LIN {X 0,Y 257.714,Z 380.293,A -85,B 0,C 180,E1 -18614.986,E2 -18614.986} C_VEL
LIN {X 0,Y 256.37,Z 386.255,A -85,B 0,C 180,E1 -18617.333,E2 -18617.333} C_VEL
LIN {X 0,Y 255.344,Z 390.968,A -85,B 0,C 180,E1 -18619.695,E2 -18619.695} C_VEL
LIN {X 0,Y 254.63,Z 394.575,A -85,B 0,C 180,E1 -18622.069,E2 -18622.069} C_VEL
LIN {X 0,Y 254.242,Z 397.09,A -85,B 0,C 180,E1 -18624.356,E2 -18624.356} C_VEL
LIN {X 0,Y 254.025,Z 398.836,A -85,B 0,C 180,E1 -18626.829,E2 -18626.829} C_VEL
LIN {X 0,Y 253.97,Z 399.449,A -85,B 0,C 180,E1 -18628.415,E2 -18628.415} C_VEL
LIN {X 0,Y 253.984,Z 399.68,A -85,B 0,C 180,E1 -18630.001,E2 -18630.001} C_VEL
LIN {X 0,Y 253.969,Z 399.486,A -85,B 0,C 180,E1 -18631.586,E2 -18631.586} C_VEL
LIN {X 0,Y 254.023,Z 398.897,A -85,B 0,C 180,E1 -18633.173,E2 -18633.173} C_VEL
LIN {X 0,Y 254.332,Z 396.56,A -85,B 0,C 180,E1 -18636.347,E2 -18636.347} C_VEL
LIN {X 0,Y 254.856,Z 393.678,A -85,B 0,C 180,E1 -18638.724,E2 -18638.724} C_VEL
LIN {X 0,Y 255.623,Z 389.771,A -85,B 0,C 180,E1 -18641.097,E2 -18641.097} C_VEL
LIN {X 0,Y 256.754,Z 384.732,A -85,B 0,C 180,E1 -18643.454,E2 -18643.454} C_VEL
LIN {X 0,Y 258.236,Z 378.388,A -85,B 0,C 180,E1 -18645.793,E2 -18645.793} C_VEL
LIN {X 0,Y 260.119,Z 370.451,A -85,B 0,C 180,E1 -18648.102,E2 -18648.102} C_VEL
LIN {X 0,Y 262.191,Z 360.583,A -85,B 0,C 180,E1 -18650.394,E2 -18650.394} C_VEL
LIN {X 0,Y 264.233,Z 350.223,A -85,B 0,C 180,E1 -18652.273,E2 -18652.273} C_VEL
LIN {X 0,Y 266.512,Z 338.538,A -85,B 0,C 180,E1 -18653.919,E2 -18653.919} C_VEL
LIN {X 0,Y 268.291,Z 326.889,A -85,B 0,C 180,E1 -18655.194,E2 -18655.194} C_VEL
LIN {X 0,Y 269.794,Z 314.77,A -85,B 0,C 180,E1 -18656.181,E2 -18656.181} C_VEL
LIN {X 0,Y 270.995,Z 301.535,A -85,B 0,C 180,E1 -18656.939,E2 -18656.939} C_VEL
LIN {X 0,Y 271.629,Z 288.539,A -85,B 0,C 180,E1 -18657.391,E2 -18657.391} C_VEL
LIN {X 0,Y 273.449,Z 229.394,A -85,B 0,C 180,E1 -18658.918,E2 -18658.918} C_VEL
LIN {X 0,Y 271.728,Z 220.396,A -85,B 0,C 180,E1 -18659.386,E2 -18659.386} C_VEL
LIN {X 0,Y 264.81,Z 203.367,A -85,B 0,C 180,E1 -18660.76,E2 -18660.76} C_VEL
LIN {X 0,Y 257.854,Z 188.654,A -85,B 0,C 180,E1 -18662.208,E2 -18662.208} C_VEL
LIN {X 0,Y 256.723,Z 184.121,A -85,B 0,C 180,E1 -18664.077,E2 -18664.077} C_VEL
LIN {X 0,Y 256.131,Z 181.593,A -85,B 0,C 180,E1 -18665.365,E2 -18665.365} C_VEL
LIN {X 0,Y 256.072,Z 181.56,A -85,B 0,C 180,E1 -18669.142,E2 -18669.142} C_VEL
LIN {X 0,Y 256.062,Z 181.59,A -85,B 0,C 180,E1 -18673.327,E2 -18673.327} C_VEL
LIN {X 0,Y 256.069,Z 181.556,A -85,B 0,C 180,E1 -18677.819,E2 -18677.819} C_VEL
LIN {X 0,Y 256.071,Z 181.588,A -85,B 0,C 180,E1 -18680.858,E2 -18680.858} C_VEL
LIN {X 0,Y 256.13,Z 181.548,A -85,B 0,C 180,E1 -18682.867,E2 -18682.867} C_VEL
LIN {X 0,Y 256.067,Z 181.55,A -85,B 0,C 180,E1 -18686.707,E2 -18686.707} C_VEL
LIN {X 0,Y 256.113,Z 181.58,A -85,B 0,C 180,E1 -18690.4,E2 -18690.4} C_VEL
LIN {X 0,Y 256.169,Z 181.575,A -85,B 0,C 180,E1 -18694.87,E2 -18694.87} C_VEL
LIN {X 0,Y 256.16,Z 181.565,A -85,B 0,C 180,E1 -18699.104,E2 -18699.104} C_VEL
LIN {X 0,Y 256.277,Z 181.542,A -85,B 0,C 180,E1 -18704.083,E2 -18704.083} C_VEL
LIN {X 0,Y 256.307,Z 181.551,A -85,B 0,C 180,E1 -18708.934,E2 -18708.934} C_VEL
LIN {X 0,Y 256.537,Z 181.514,A -85,B 0,C 180,E1 -18712.127,E2 -18712.127} C_VEL
LIN {X 0,Y 256.5,Z 181.515,A -85,B 0,C 180,E1 -18716.974,E2 -18716.974} C_VEL
LIN {X 0,Y 255.921,Z 181.588,A -85,B 0,C 180,E1 -18718.288,E2 -18718.288} C_VEL
LIN {X 0,Y 254.374,Z 181.792,A -85,B 0,C 180,E1 -18719.578,E2 -18719.578} C_VEL
LIN {X 0,Y 250.591,Z 182.267,A -85,B 0,C 180,E1 -18722.171,E2 -18722.171} C_VEL
LIN {X 0,Y 249.457,Z 182.394,A -85,B 0,C 180,E1 -18723.523,E2 -18723.523} C_VEL
LIN {X 0,Y 249.335,Z 182.405,A -85,B 0,C 180,E1 -18723.982,E2 -18723.982} C_VEL
LIN {X 0,Y 249.439,Z 182.413,A -85,B 0,C 180,E1 -18728.099,E2 -18728.099} C_VEL
LIN {X 0,Y 249.185,Z 182.436,A -85,B 0,C 180,E1 -18733.04,E2 -18733.04} C_VEL
LIN {X 0,Y 249.194,Z 182.434,A -85,B 0,C 180,E1 -18736.486,E2 -18736.486} C_VEL
LIN {X 0,Y 249.079,Z 182.457,A -85,B 0,C 180,E1 -18741.519,E2 -18741.519} C_VEL
LIN {X 0,Y 249.115,Z 182.447,A -85,B 0,C 180,E1 -18745.475,E2 -18745.475} C_VEL
LIN {X 0,Y 249.071,Z 182.447,A -85,B 0,C 180,E1 -18748.989,E2 -18748.989} C_VEL
LIN {X 0,Y 249.029,Z 182.466,A -85,B 0,C 180,E1 -18752.426,E2 -18752.426} C_VEL
LIN {X 0,Y 249.028,Z 182.415,A -85,B 0,C 180,E1 -18756.346,E2 -18756.346} C_VEL
LIN {X 0,Y 249.005,Z 182.468,A -85,B 0,C 180,E1 -18760.478,E2 -18760.478} C_VEL
LIN {X 0,Y 248.986,Z 182.47,A -85,B 0,C 180,E1 -18764.883,E2 -18764.883} C_VEL
LIN {X 0,Y 249.009,Z 182.459,A -85,B 0,C 180,E1 -18767.362,E2 -18767.362} C_VEL
LIN {X 0,Y 249.027,Z 182.436,A -85,B 0,C 180,E1 -18771.62,E2 -18771.62} C_VEL
LIN {X 0,Y 249.101,Z 182.673,A -85,B 0,C 180,E1 -18772.58,E2 -18772.58} C_VEL
LIN {X 0,Y 251.278,Z 191.568,A -85,B 0,C 180,E1 -18776.62,E2 -18776.62} C_VEL
LIN {X 0,Y 251.564,Z 192.641,A -85,B 0,C 180,E1 -18776.942,E2 -18776.942} C_VEL
LIN {X 0,Y 259.446,Z 209.734,A -85,B 0,C 180,E1 -18778.65,E2 -18778.65} C_VEL
LIN {X 0,Y 264.513,Z 222.59,A -85,B 0,C 180,E1 -18779.712,E2 -18779.712} C_VEL
LIN {X 0,Y 267.062,Z 239.045,A -85,B 0,C 180,E1 -18780.529,E2 -18780.529} C_VEL
LIN {X 0,Y 264.966,Z 300.538,A -85,B 0,C 180,E1 -18782.182,E2 -18782.182} C_VEL
LIN {X 0,Y 263.782,Z 314.425,A -85,B 0,C 180,E1 -18782.854,E2 -18782.854} C_VEL
LIN {X 0,Y 262.218,Z 326.85,A -85,B 0,C 180,E1 -18783.753,E2 -18783.753} C_VEL
LIN {X 0,Y 260.587,Z 337.935,A -85,B 0,C 180,E1 -18784.863,E2 -18784.863} C_VEL
LIN {X 0,Y 258.448,Z 349.485,A -85,B 0,C 180,E1 -18786.353,E2 -18786.353} C_VEL
LIN {X 0,Y 256.294,Z 359.884,A -85,B 0,C 180,E1 -18788.061,E2 -18788.061} C_VEL
LIN {X 0,Y 254.189,Z 369.509,A -85,B 0,C 180,E1 -18790.062,E2 -18790.062} C_VEL
LIN {X 0,Y 252.306,Z 377.598,A -85,B 0,C 180,E1 -18792.157,E2 -18792.157} C_VEL
LIN {X 0,Y 250.517,Z 385.001,A -85,B 0,C 180,E1 -18794.543,E2 -18794.543} C_VEL
LIN {X 0,Y 249.061,Z 390.944,A -85,B 0,C 180,E1 -18796.953,E2 -18796.953} C_VEL
LIN {X 0,Y 248.039,Z 395.639,A -85,B 0,C 180,E1 -18799.387,E2 -18799.387} C_VEL
LIN {X 0,Y 247.375,Z 399.225,A -85,B 0,C 180,E1 -18801.833,E2 -18801.833} C_VEL
LIN {X 0,Y 247.084,Z 401.074,A -85,B 0,C 180,E1 -18803.466,E2 -18803.466} C_VEL
LIN {X 0,Y 246.923,Z 402.459,A -85,B 0,C 180,E1 -18805.101,E2 -18805.101} C_VEL
LIN {X 0,Y 246.86,Z 404.051,A -85,B 0,C 180,E1 -18808.368,E2 -18808.368} C_VEL
LIN {X 0,Y 246.891,Z 404.262,A -85,B 0,C 180,E1 -18809.999,E2 -18809.999} C_VEL
LIN {X 0,Y 246.86,Z 404.041,A -85,B 0,C 180,E1 -18811.631,E2 -18811.631} C_VEL
LIN {X 0,Y 246.924,Z 402.437,A -85,B 0,C 180,E1 -18814.897,E2 -18814.897} C_VEL
LIN {X 0,Y 247.086,Z 401.042,A -85,B 0,C 180,E1 -18816.532,E2 -18816.532} C_VEL
LIN {X 0,Y 247.563,Z 398.112,A -85,B 0,C 180,E1 -18818.982,E2 -18818.982} C_VEL
LIN {X 0,Y 248.329,Z 394.147,A -85,B 0,C 180,E1 -18821.425,E2 -18821.425} C_VEL
LIN {X 0,Y 249.704,Z 388.048,A -85,B 0,C 180,E1 -18824.256,E2 -18824.256} C_VEL
LIN {X 0,Y 251.396,Z 381.387,A -85,B 0,C 180,E1 -18826.65,E2 -18826.65} C_VEL
LIN {X 0,Y 253.374,Z 373.12,A -85,B 0,C 180,E1 -18829.02,E2 -18829.02} C_VEL
LIN {X 0,Y 255.181,Z 364.638,A -85,B 0,C 180,E1 -18830.978,E2 -18830.978} C_VEL
LIN {X 0,Y 257.424,Z 354.157,A -85,B 0,C 180,E1 -18832.894,E2 -18832.894} C_VEL
LIN {X 0,Y 259.694,Z 342.355,A -85,B 0,C 180,E1 -18834.586,E2 -18834.586} C_VEL
LIN {X 0,Y 261.675,Z 330.462,A -85,B 0,C 180,E1 -18835.875,E2 -18835.875} C_VEL
LIN {X 0,Y 263.243,Z 318.078,A -85,B 0,C 180,E1 -18836.883,E2 -18836.883} C_VEL
LIN {X 0,Y 264.56,Z 305.317,A -85,B 0,C 180,E1 -18837.594,E2 -18837.594} C_VEL
LIN {X 0,Y 265.264,Z 291.803,A -85,B 0,C 180,E1 -18838.051,E2 -18838.051} C_VEL
LIN {X 0,Y 266.926,Z 237.825,A -85,B 0,C 180,E1 -18839.482,E2 -18839.482} C_VEL
LIN {X 0,Y 264.151,Z 221.481,A -85,B 0,C 180,E1 -18840.324,E2 -18840.324} C_VEL
LIN {X 0,Y 257.7,Z 205.912,A -85,B 0,C 180,E1 -18841.661,E2 -18841.661} C_VEL
LIN {X 0,Y 251.481,Z 192.518,A -85,B 0,C 180,E1 -18843.029,E2 -18843.029} C_VEL
LIN {X 0,Y 250.518,Z 188.305,A -85,B 0,C 180,E1 -18844.751,E2 -18844.751} C_VEL
LIN {X 0,Y 249.06,Z 182.485,A -85,B 0,C 180,E1 -18847.542,E2 -18847.542} C_VEL
LIN {X 0,Y 249.002,Z 182.46,A -85,B 0,C 180,E1 -18850.477,E2 -18850.477} C_VEL
LIN {X 0,Y 248.981,Z 182.473,A -85,B 0,C 180,E1 -18854.882,E2 -18854.882} C_VEL
LIN {X 0,Y 249.004,Z 182.457,A -85,B 0,C 180,E1 -18857.36,E2 -18857.36} C_VEL
LIN {X 0,Y 249.02,Z 182.43,A -85,B 0,C 180,E1 -18861.618,E2 -18861.618} C_VEL
LIN {X 0,Y 249.037,Z 182.439,A -85,B 0,C 180,E1 -18865.638,E2 -18865.638} C_VEL
LIN {X 0,Y 249.041,Z 182.454,A -85,B 0,C 180,E1 -18869.472,E2 -18869.472} C_VEL
LIN {X 0,Y 249.061,Z 182.462,A -85,B 0,C 180,E1 -18873.161,E2 -18873.161} C_VEL
LIN {X 0,Y 249.052,Z 182.447,A -85,B 0,C 180,E1 -18876.73,E2 -18876.73} C_VEL
LIN {X 0,Y 249.082,Z 182.452,A -85,B 0,C 180,E1 -18880.209,E2 -18880.209} C_VEL
LIN {X 0,Y 249.188,Z 182.437,A -85,B 0,C 180,E1 -18883.618,E2 -18883.618} C_VEL
LIN {X 0,Y 249.243,Z 182.418,A -85,B 0,C 180,E1 -18888.616,E2 -18888.616} C_VEL
LIN {X 0,Y 249.471,Z 182.409,A -85,B 0,C 180,E1 -18891.903,E2 -18891.903} C_VEL
LIN {X 0,Y 249.422,Z 182.401,A -85,B 0,C 180,E1 -18896.769,E2 -18896.769} C_VEL
LIN {X 0,Y 249.719,Z 182.375,A -85,B 0,C 180,E1 -18900,E2 -18900} C_VEL
LIN {X 0,Y 249.423,Z 182.397,A -85,B 0,C 180,E1 -18903.231,E2 -18903.231} C_VEL
LIN {X 0,Y 249.473,Z 182.391,A -85,B 0,C 180,E1 -18908.098,E2 -18908.098} C_VEL
LIN {X 0,Y 249.244,Z 182.433,A -85,B 0,C 180,E1 -18911.384,E2 -18911.384} C_VEL
LIN {X 0,Y 249.211,Z 182.424,A -85,B 0,C 180,E1 -18916.504,E2 -18916.504} C_VEL
LIN {X 0,Y 249.08,Z 182.443,A -85,B 0,C 180,E1 -18921.519,E2 -18921.519} C_VEL
LIN {X 0,Y 249.124,Z 182.453,A -85,B 0,C 180,E1 -18925.483,E2 -18925.483} C_VEL
LIN {X 0,Y 249.077,Z 182.451,A -85,B 0,C 180,E1 -18928.994,E2 -18928.994} C_VEL
LIN {X 0,Y 249.024,Z 182.447,A -85,B 0,C 180,E1 -18932.427,E2 -18932.427} C_VEL
LIN {X 0,Y 249.024,Z 182.418,A -85,B 0,C 180,E1 -18936.347,E2 -18936.347} C_VEL
LIN {X 0,Y 249.001,Z 182.465,A -85,B 0,C 180,E1 -18940.479,E2 -18940.479} C_VEL
LIN {X 0,Y 248.988,Z 182.442,A -85,B 0,C 180,E1 -18944.883,E2 -18944.883} C_VEL
LIN {X 0,Y 249.012,Z 182.465,A -85,B 0,C 180,E1 -18947.364,E2 -18947.364} C_VEL
LIN {X 0,Y 249.041,Z 182.452,A -85,B 0,C 180,E1 -18952.202,E2 -18952.202} C_VEL
LIN {X 0,Y 249.12,Z 182.674,A -85,B 0,C 180,E1 -18954.191,E2 -18954.191} C_VEL
LIN {X 0,Y 250.596,Z 188.64,A -85,B 0,C 180,E1 -18956.872,E2 -18956.872} C_VEL
LIN {X 0,Y 257.409,Z 202.804,A -85,B 0,C 180,E1 -18958.373,E2 -18958.373} C_VEL
LIN {X 0,Y 263.323,Z 216.402,A -85,B 0,C 180,E1 -18959.587,E2 -18959.587} C_VEL
LIN {X 0,Y 266.09,Z 223.996,A -85,B 0,C 180,E1 -18960.17,E2 -18960.17} C_VEL
LIN {X 0,Y 267.251,Z 231.184,A -85,B 0,C 180,E1 -18960.531,E2 -18960.531} C_VEL
LIN {X 0,Y 265.118,Z 295.563,A -85,B 0,C 180,E1 -18962.255,E2 -18962.255} C_VEL
LIN {X 0,Y 263.939,Z 308.907,A -85,B 0,C 180,E1 -18962.873,E2 -18962.873} C_VEL
LIN {X 0,Y 262.584,Z 321.658,A -85,B 0,C 180,E1 -18963.794,E2 -18963.794} C_VEL
LIN {X 0,Y 260.868,Z 332.985,A -85,B 0,C 180,E1 -18964.894,E2 -18964.894} C_VEL
LIN {X 0,Y 258.791,Z 344.638,A -85,B 0,C 180,E1 -18966.388,E2 -18966.388} C_VEL
LIN {X 0,Y 256.651,Z 355.106,A -85,B 0,C 180,E1 -18968.094,E2 -18968.094} C_VEL
LIN {X 0,Y 254.961,Z 363.35,A -85,B 0,C 180,E1 -18969.773,E2 -18969.773} C_VEL
LIN {X 0,Y 253.136,Z 371.541,A -85,B 0,C 180,E1 -18971.801,E2 -18971.801} C_VEL
LIN {X 0,Y 251.114,Z 379.246,A -85,B 0,C 180,E1 -18974.166,E2 -18974.166} C_VEL
LIN {X 0,Y 249.445,Z 386.321,A -85,B 0,C 180,E1 -18976.975,E2 -18976.975} C_VEL
LIN {X 0,Y 248.333,Z 391.034,A -85,B 0,C 180,E1 -18979.401,E2 -18979.401} C_VEL
LIN {X 0,Y 247.602,Z 394.641,A -85,B 0,C 180,E1 -18981.842,E2 -18981.842} C_VEL
LIN {X 0,Y 247.138,Z 397.385,A -85,B 0,C 180,E1 -18984.453,E2 -18984.453} C_VEL
LIN {X 0,Y 246.931,Z 398.901,A -85,B 0,C 180,E1 -18986.738,E2 -18986.738} C_VEL
LIN {X 0,Y 246.884,Z 399.514,A -85,B 0,C 180,E1 -18988.369,E2 -18988.369} C_VEL
LIN {X 0,Y 246.894,Z 399.745,A -85,B 0,C 180,E1 -18990.001,E2 -18990.001} C_VEL
LIN {X 0,Y 246.883,Z 399.551,A -85,B 0,C 180,E1 -18991.632,E2 -18991.632} C_VEL
LIN {X 0,Y 247.06,Z 397.989,A -85,B 0,C 180,E1 -18994.896,E2 -18994.896} C_VEL
LIN {X 0,Y 247.268,Z 396.624,A -85,B 0,C 180,E1 -18996.529,E2 -18996.529} C_VEL
LIN {X 0,Y 247.831,Z 393.742,A -85,B 0,C 180,E1 -18998.973,E2 -18998.973} C_VEL
LIN {X 0,Y 248.63,Z 389.835,A -85,B 0,C 180,E1 -19001.413,E2 -19001.413} C_VEL
LIN {X 0,Y 249.818,Z 384.795,A -85,B 0,C 180,E1 -19003.835,E2 -19003.835} C_VEL
LIN {X 0,Y 251.39,Z 378.451,A -85,B 0,C 180,E1 -19006.235,E2 -19006.235} C_VEL
LIN {X 0,Y 253.358,Z 370.514,A -85,B 0,C 180,E1 -19008.603,E2 -19008.603} C_VEL
LIN {X 0,Y 255.273,Z 361.785,A -85,B 0,C 180,E1 -19010.702,E2 -19010.702} C_VEL
LIN {X 0,Y 257.45,Z 351.456,A -85,B 0,C 180,E1 -19012.681,E2 -19012.681} C_VEL
LIN {X 0,Y 259.778,Z 340.022,A -85,B 0,C 180,E1 -19014.367,E2 -19014.367} C_VEL
LIN {X 0,Y 261.58,Z 328.795,A -85,B 0,C 180,E1 -19015.673,E2 -19015.673} C_VEL
LIN {X 0,Y 263.165,Z 317.39,A -85,B 0,C 180,E1 -19016.679,E2 -19016.679} C_VEL
LIN {X 0,Y 264.491,Z 304.333,A -85,B 0,C 180,E1 -19017.496,E2 -19017.496} C_VEL
LIN {X 0,Y 265.285,Z 291.804,A -85,B 0,C 180,E1 -19017.996,E2 -19017.996} C_VEL
LIN {X 0,Y 267.208,Z 230.204,A -85,B 0,C 180,E1 -19019.637,E2 -19019.637} C_VEL
LIN {X 0,Y 265.891,Z 223.22,A -85,B 0,C 180,E1 -19020.012,E2 -19020.012} C_VEL
LIN {X 0,Y 259.258,Z 206.741,A -85,B 0,C 180,E1 -19021.387,E2 -19021.387} C_VEL
LIN {X 0,Y 251.967,Z 191.659,A -85,B 0,C 180,E1 -19022.906,E2 -19022.906} C_VEL
LIN {X 0,Y 250.562,Z 188.505,A -85,B 0,C 180,E1 -19023.302,E2 -19023.302} C_VEL
LIN {X 0,Y 249.124,Z 182.53,A -85,B 0,C 180,E1 -19026.075,E2 -19026.075} C_VEL
LIN {X 0,Y 248.992,Z 182.437,A -85,B 0,C 180,E1 -19030.481,E2 -19030.481} C_VEL
LIN {X 0,Y 249.009,Z 182.465,A -85,B 0,C 180,E1 -19032.792,E2 -19032.792} C_VEL
LIN {X 0,Y 249.009,Z 182.431,A -85,B 0,C 180,E1 -19037.361,E2 -19037.361} C_VEL
LIN {X 0,Y 249.025,Z 182.458,A -85,B 0,C 180,E1 -19041.619,E2 -19041.619} C_VEL
LIN {X 0,Y 249.042,Z 182.411,A -85,B 0,C 180,E1 -19045.639,E2 -19045.639} C_VEL
LIN {X 0,Y 249.051,Z 182.462,A -85,B 0,C 180,E1 -19049.473,E2 -19049.473} C_VEL
LIN {X 0,Y 249.068,Z 182.448,A -85,B 0,C 180,E1 -19053.161,E2 -19053.161} C_VEL
LIN {X 0,Y 249.059,Z 182.452,A -85,B 0,C 180,E1 -19056.73,E2 -19056.73} C_VEL
LIN {X 0,Y 249.106,Z 182.453,A -85,B 0,C 180,E1 -19060.211,E2 -19060.211} C_VEL
LIN {X 0,Y 249.221,Z 182.422,A -85,B 0,C 180,E1 -19063.62,E2 -19063.62} C_VEL
LIN {X 0,Y 249.25,Z 182.432,A -85,B 0,C 180,E1 -19068.616,E2 -19068.616} C_VEL
LIN {X 0,Y 249.479,Z 182.39,A -85,B 0,C 180,E1 -19071.903,E2 -19071.903} C_VEL
LIN {X 0,Y 249.428,Z 182.397,A -85,B 0,C 180,E1 -19076.769,E2 -19076.769} C_VEL
LIN {X 0,Y 249.717,Z 182.375,A -85,B 0,C 180,E1 -19080,E2 -19080} C_VEL
LIN {X 0,Y 249.426,Z 182.401,A -85,B 0,C 180,E1 -19083.23,E2 -19083.23} C_VEL
LIN {X 0,Y 249.335,Z 182.405,A -85,B 0,C 180,E1 -19083.982,E2 -19083.982} C_VEL
LIN {X 0,Y 248.59,Z 182.501,A -85,B 0,C 180,E1 -19085.332,E2 -19085.332} C_VEL
LIN {X 0,Y 245.714,Z 182.877,A -85,B 0,C 180,E1 -19087.533,E2 -19087.533} C_VEL
LIN {X 0,Y 243.307,Z 183.171,A -85,B 0,C 180,E1 -19089.325,E2 -19089.325} C_VEL
LIN {X 0,Y 242.262,Z 183.289,A -85,B 0,C 180,E1 -19090.714,E2 -19090.714} C_VEL
LIN {X 0,Y 242.167,Z 183.299,A -85,B 0,C 180,E1 -19091.185,E2 -19091.185} C_VEL
LIN {X 0,Y 242.136,Z 183.324,A -85,B 0,C 180,E1 -19095.143,E2 -19095.143} C_VEL
LIN {X 0,Y 242.051,Z 183.317,A -85,B 0,C 180,E1 -19098.626,E2 -19098.626} C_VEL
LIN {X 0,Y 242.003,Z 183.336,A -85,B 0,C 180,E1 -19102.181,E2 -19102.181} C_VEL
LIN {X 0,Y 242.065,Z 183.33,A -85,B 0,C 180,E1 -19105.838,E2 -19105.838} C_VEL
LIN {X 0,Y 242.006,Z 183.326,A -85,B 0,C 180,E1 -19109.583,E2 -19109.583} C_VEL
LIN {X 0,Y 241.979,Z 183.332,A -85,B 0,C 180,E1 -19113.493,E2 -19113.493} C_VEL
LIN {X 0,Y 241.985,Z 183.296,A -85,B 0,C 180,E1 -19117.583,E2 -19117.583} C_VEL
LIN {X 0,Y 241.933,Z 183.341,A -85,B 0,C 180,E1 -19121.923,E2 -19121.923} C_VEL
LIN {X 0,Y 241.925,Z 183.341,A -85,B 0,C 180,E1 -19126.574,E2 -19126.574} C_VEL
LIN {X 0,Y 241.974,Z 183.334,A -85,B 0,C 180,E1 -19131.409,E2 -19131.409} C_VEL
LIN {X 0,Y 242.165,Z 184.198,A -85,B 0,C 180,E1 -19132.057,E2 -19132.057} C_VEL
LIN {X 0,Y 244.206,Z 192.08,A -85,B 0,C 180,E1 -19135.73,E2 -19135.73} C_VEL
LIN {X 0,Y 245.754,Z 195.601,A -85,B 0,C 180,E1 -19136.203,E2 -19136.203} C_VEL
LIN {X 0,Y 253.217,Z 211.541,A -85,B 0,C 180,E1 -19137.848,E2 -19137.848} C_VEL
LIN {X 0,Y 258.524,Z 224.654,A -85,B 0,C 180,E1 -19139,E2 -19139} C_VEL
LIN {X 0,Y 260.875,Z 239.859,A -85,B 0,C 180,E1 -19139.785,E2 -19139.785} C_VEL
LIN {X 0,Y 258.719,Z 300.487,A -85,B 0,C 180,E1 -19141.45,E2 -19141.45} C_VEL
LIN {X 0,Y 257.502,Z 314.37,A -85,B 0,C 180,E1 -19142.135,E2 -19142.135} C_VEL
LIN {X 0,Y 255.862,Z 326.791,A -85,B 0,C 180,E1 -19143.049,E2 -19143.049} C_VEL
LIN {X 0,Y 254.18,Z 337.874,A -85,B 0,C 180,E1 -19144.184,E2 -19144.184} C_VEL
LIN {X 0,Y 251.961,Z 349.424,A -85,B 0,C 180,E1 -19145.706,E2 -19145.706} C_VEL
LIN {X 0,Y 249.696,Z 359.822,A -85,B 0,C 180,E1 -19147.45,E2 -19147.45} C_VEL
LIN {X 0,Y 247.752,Z 368.326,A -85,B 0,C 180,E1 -19149.232,E2 -19149.232} C_VEL
LIN {X 0,Y 245.894,Z 376.164,A -85,B 0,C 180,E1 -19151.244,E2 -19151.244} C_VEL
LIN {X 0,Y 243.934,Z 383.82,A -85,B 0,C 180,E1 -19153.685,E2 -19153.685} C_VEL
LIN {X 0,Y 242.11,Z 390.88,A -85,B 0,C 180,E1 -19156.571,E2 -19156.571} C_VEL
LIN {X 0,Y 241.027,Z 395.575,A -85,B 0,C 180,E1 -19159.074,E2 -19159.074} C_VEL
LIN {X 0,Y 240.328,Z 399.161,A -85,B 0,C 180,E1 -19161.592,E2 -19161.592} C_VEL
LIN {X 0,Y 240.031,Z 401.009,A -85,B 0,C 180,E1 -19163.274,E2 -19163.274} C_VEL
LIN {X 0,Y 239.836,Z 402.478,A -85,B 0,C 180,E1 -19165.081,E2 -19165.081} C_VEL
LIN {X 0,Y 239.773,Z 403.987,A -85,B 0,C 180,E1 -19168.32,E2 -19168.32} C_VEL
LIN {X 0,Y 239.804,Z 404.197,A -85,B 0,C 180,E1 -19169.999,E2 -19169.999} C_VEL
LIN {X 0,Y 239.774,Z 403.976,A -85,B 0,C 180,E1 -19171.679,E2 -19171.679} C_VEL
LIN {X 0,Y 239.844,Z 402.372,A -85,B 0,C 180,E1 -19175.042,E2 -19175.042} C_VEL
LIN {X 0,Y 240.033,Z 400.976,A -85,B 0,C 180,E1 -19176.725,E2 -19176.725} C_VEL
LIN {X 0,Y 240.542,Z 398.046,A -85,B 0,C 180,E1 -19179.246,E2 -19179.246} C_VEL
LIN {X 0,Y 241.344,Z 394.08,A -85,B 0,C 180,E1 -19181.761,E2 -19181.761} C_VEL
LIN {X 0,Y 242.787,Z 387.981,A -85,B 0,C 180,E1 -19184.671,E2 -19184.671} C_VEL
LIN {X 0,Y 244.598,Z 381.32,A -85,B 0,C 180,E1 -19187.127,E2 -19187.127} C_VEL
LIN {X 0,Y 246.664,Z 373.053,A -85,B 0,C 180,E1 -19189.558,E2 -19189.558} C_VEL
LIN {X 0,Y 248.534,Z 364.57,A -85,B 0,C 180,E1 -19191.567,E2 -19191.567} C_VEL
LIN {X 0,Y 250.886,Z 354.089,A -85,B 0,C 180,E1 -19193.526,E2 -19193.526} C_VEL
LIN {X 0,Y 253.26,Z 342.286,A -85,B 0,C 180,E1 -19195.254,E2 -19195.254} C_VEL
LIN {X 0,Y 255.3,Z 330.391,A -85,B 0,C 180,E1 -19196.571,E2 -19196.571} C_VEL
LIN {X 0,Y 256.939,Z 318.005,A -85,B 0,C 180,E1 -19197.598,E2 -19197.598} C_VEL
LIN {X 0,Y 258.3,Z 305.24,A -85,B 0,C 180,E1 -19198.322,E2 -19198.322} C_VEL
LIN {X 0,Y 259.029,Z 291.717,A -85,B 0,C 180,E1 -19198.788,E2 -19198.788} C_VEL
LIN {X 0,Y 260.752,Z 239.019,A -85,B 0,C 180,E1 -19200.212,E2 -19200.212} C_VEL
LIN {X 0,Y 258.277,Z 224.097,A -85,B 0,C 180,E1 -19201.003,E2 -19201.003} C_VEL
LIN {X 0,Y 252.02,Z 208.973,A -85,B 0,C 180,E1 -19202.357,E2 -19202.357} C_VEL
LIN {X 0,Y 245.469,Z 195.187,A -85,B 0,C 180,E1 -19203.802,E2 -19203.802} C_VEL
LIN {X 0,Y 244.197,Z 192.213,A -85,B 0,C 180,E1 -19204.192,E2 -19204.192} C_VEL
LIN {X 0,Y 242.403,Z 184.961,A -85,B 0,C 180,E1 -19207.505,E2 -19207.505} C_VEL
LIN {X 0,Y 241.989,Z 183.354,A -85,B 0,C 180,E1 -19208.424,E2 -19208.424} C_VEL
LIN {X 0,Y 241.929,Z 183.344,A -85,B 0,C 180,E1 -19211.922,E2 -19211.922} C_VEL
LIN {X 0,Y 241.92,Z 183.338,A -85,B 0,C 180,E1 -19216.572,E2 -19216.572} C_VEL
LIN {X 0,Y 241.951,Z 183.336,A -85,B 0,C 180,E1 -19220.28,E2 -19220.28} C_VEL
LIN {X 0,Y 241.975,Z 183.299,A -85,B 0,C 180,E1 -19224.487,E2 -19224.487} C_VEL
LIN {X 0,Y 241.967,Z 183.345,A -85,B 0,C 180,E1 -19228.479,E2 -19228.479} C_VEL
LIN {X 0,Y 241.994,Z 183.338,A -85,B 0,C 180,E1 -19232.311,E2 -19232.311} C_VEL
LIN {X 0,Y 242.033,Z 183.318,A -85,B 0,C 180,E1 -19236.013,E2 -19236.013} C_VEL
LIN {X 0,Y 242.016,Z 183.337,A -85,B 0,C 180,E1 -19239.606,E2 -19239.606} C_VEL
LIN {X 0,Y 242.12,Z 183.312,A -85,B 0,C 180,E1 -19243.306,E2 -19243.306} C_VEL
LIN {X 0,Y 242.176,Z 183.298,A -85,B 0,C 180,E1 -19248.279,E2 -19248.279} C_VEL
LIN {X 0,Y 242.418,Z 183.287,A -85,B 0,C 180,E1 -19251.665,E2 -19251.665} C_VEL
LIN {X 0,Y 242.245,Z 183.287,A -85,B 0,C 180,E1 -19255.007,E2 -19255.007} C_VEL
LIN {X 0,Y 242.626,Z 183.262,A -85,B 0,C 180,E1 -19258.34,E2 -19258.34} C_VEL
LIN {X 0,Y 242.626,Z 183.242,A -85,B 0,C 180,E1 -19261.66,E2 -19261.66} C_VEL
LIN {X 0,Y 242.414,Z 183.282,A -85,B 0,C 180,E1 -19266.815,E2 -19266.815} C_VEL
LIN {X 0,Y 242.306,Z 183.28,A -85,B 0,C 180,E1 -19270.022,E2 -19270.022} C_VEL
LIN {X 0,Y 242.156,Z 183.302,A -85,B 0,C 180,E1 -19275.142,E2 -19275.142} C_VEL
LIN {X 0,Y 242.066,Z 183.333,A -85,B 0,C 180,E1 -19278.625,E2 -19278.625} C_VEL
LIN {X 0,Y 242.006,Z 183.322,A -85,B 0,C 180,E1 -19282.181,E2 -19282.181} C_VEL
LIN {X 0,Y 242.06,Z 183.33,A -85,B 0,C 180,E1 -19285.839,E2 -19285.839} C_VEL
LIN {X 0,Y 242.024,Z 183.334,A -85,B 0,C 180,E1 -19289.581,E2 -19289.581} C_VEL
LIN {X 0,Y 241.975,Z 183.302,A -85,B 0,C 180,E1 -19293.494,E2 -19293.494} C_VEL
LIN {X 0,Y 241.981,Z 183.314,A -85,B 0,C 180,E1 -19297.584,E2 -19297.584} C_VEL
LIN {X 0,Y 241.929,Z 183.321,A -85,B 0,C 180,E1 -19301.925,E2 -19301.925} C_VEL
LIN {X 0,Y 241.929,Z 183.35,A -85,B 0,C 180,E1 -19306.573,E2 -19306.573} C_VEL
LIN {X 0,Y 241.993,Z 183.319,A -85,B 0,C 180,E1 -19311.642,E2 -19311.642} C_VEL
LIN {X 0,Y 242.064,Z 183.552,A -85,B 0,C 180,E1 -19313.337,E2 -19313.337} C_VEL
LIN {X 0,Y 243.357,Z 188.803,A -85,B 0,C 180,E1 -19315.768,E2 -19315.768} C_VEL
LIN {X 0,Y 249.859,Z 201.93,A -85,B 0,C 180,E1 -19317.268,E2 -19317.268} C_VEL
LIN {X 0,Y 256.236,Z 216.029,A -85,B 0,C 180,E1 -19318.637,E2 -19318.637} C_VEL
LIN {X 0,Y 260.178,Z 226.549,A -85,B 0,C 180,E1 -19319.498,E2 -19319.498} C_VEL
LIN {X 0,Y 261.071,Z 232.307,A -85,B 0,C 180,E1 -19319.794,E2 -19319.794} C_VEL
LIN {X 0,Y 258.877,Z 295.646,A -85,B 0,C 180,E1 -19321.526,E2 -19321.526} C_VEL
LIN {X 0,Y 257.656,Z 308.982,A -85,B 0,C 180,E1 -19322.154,E2 -19322.154} C_VEL
LIN {X 0,Y 256.243,Z 321.73,A -85,B 0,C 180,E1 -19323.094,E2 -19323.094} C_VEL
LIN {X 0,Y 254.448,Z 333.055,A -85,B 0,C 180,E1 -19324.215,E2 -19324.215} C_VEL
LIN {X 0,Y 252.289,Z 344.707,A -85,B 0,C 180,E1 -19325.741,E2 -19325.741} C_VEL
LIN {X 0,Y 250.08,Z 355.174,A -85,B 0,C 180,E1 -19327.488,E2 -19327.488} C_VEL
LIN {X 0,Y 248.162,Z 364.038,A -85,B 0,C 180,E1 -19329.345,E2 -19329.345} C_VEL
LIN {X 0,Y 246.025,Z 372.998,A -85,B 0,C 180,E1 -19331.687,E2 -19331.687} C_VEL
LIN {X 0,Y 243.983,Z 380.427,A -85,B 0,C 180,E1 -19334.12,E2 -19334.12} C_VEL
LIN {X 0,Y 242.514,Z 386.388,A -85,B 0,C 180,E1 -19336.596,E2 -19336.596} C_VEL
LIN {X 0,Y 241.341,Z 391.1,A -85,B 0,C 180,E1 -19339.09,E2 -19339.09} C_VEL
LIN {X 0,Y 240.556,Z 394.707,A -85,B 0,C 180,E1 -19341.601,E2 -19341.601} C_VEL
LIN {X 0,Y 240.025,Z 397.702,A -85,B 0,C 180,E1 -19344.583,E2 -19344.583} C_VEL
LIN {X 0,Y 239.841,Z 398.967,A -85,B 0,C 180,E1 -19346.641,E2 -19346.641} C_VEL
LIN {X 0,Y 239.8,Z 399.579,A -85,B 0,C 180,E1 -19348.321,E2 -19348.321} C_VEL
LIN {X 0,Y 239.807,Z 399.81,A -85,B 0,C 180,E1 -19350.001,E2 -19350.001} C_VEL
LIN {X 0,Y 239.799,Z 399.615,A -85,B 0,C 180,E1 -19351.68,E2 -19351.68} C_VEL
LIN {X 0,Y 239.97,Z 398.053,A -85,B 0,C 180,E1 -19355.041,E2 -19355.041} C_VEL
LIN {X 0,Y 240.205,Z 396.689,A -85,B 0,C 180,E1 -19356.721,E2 -19356.721} C_VEL
LIN {X 0,Y 240.794,Z 393.806,A -85,B 0,C 180,E1 -19359.238,E2 -19359.238} C_VEL
LIN {X 0,Y 241.661,Z 389.899,A -85,B 0,C 180,E1 -19361.746,E2 -19361.746} C_VEL
LIN {X 0,Y 242.904,Z 384.859,A -85,B 0,C 180,E1 -19364.237,E2 -19364.237} C_VEL
LIN {X 0,Y 244.571,Z 378.514,A -85,B 0,C 180,E1 -19366.7,E2 -19366.7} C_VEL
LIN {X 0,Y 246.618,Z 370.577,A -85,B 0,C 180,E1 -19369.131,E2 -19369.131} C_VEL
LIN {X 0,Y 248.56,Z 362.147,A -85,B 0,C 180,E1 -19371.214,E2 -19371.214} C_VEL
LIN {X 0,Y 250.685,Z 352.618,A -85,B 0,C 180,E1 -19373.11,E2 -19373.11} C_VEL
LIN {X 0,Y 253.017,Z 341.508,A -85,B 0,C 180,E1 -19374.843,E2 -19374.843} C_VEL
LIN {X 0,Y 255.215,Z 328.854,A -85,B 0,C 180,E1 -19376.362,E2 -19376.362} C_VEL
LIN {X 0,Y 256.984,Z 316.183,A -85,B 0,C 180,E1 -19377.484,E2 -19377.484} C_VEL
LIN {X 0,Y 258.288,Z 303.471,A -85,B 0,C 180,E1 -19378.27,E2 -19378.27} C_VEL
LIN {X 0,Y 259.107,Z 290.345,A -85,B 0,C 180,E1 -19378.78,E2 -19378.78} C_VEL
LIN {X 0,Y 261.055,Z 231.321,A -85,B 0,C 180,E1 -19380.375,E2 -19380.375} C_VEL
LIN {X 0,Y 259.856,Z 225.337,A -85,B 0,C 180,E1 -19380.718,E2 -19380.718} C_VEL
LIN {X 0,Y 253.661,Z 209.944,A -85,B 0,C 180,E1 -19382.057,E2 -19382.057} C_VEL
LIN {X 0,Y 246.715,Z 195.495,A -85,B 0,C 180,E1 -19383.568,E2 -19383.568} C_VEL
LIN {X 0,Y 243.35,Z 188.71,A -85,B 0,C 180,E1 -19384.397,E2 -19384.397} C_VEL
LIN {X 0,Y 242.076,Z 183.57,A -85,B 0,C 180,E1 -19386.801,E2 -19386.801} C_VEL
LIN {X 0,Y 241.949,Z 183.314,A -85,B 0,C 180,E1 -19389.72,E2 -19389.72} C_VEL
LIN {X 0,Y 241.926,Z 183.34,A -85,B 0,C 180,E1 -19394.203,E2 -19394.203} C_VEL
LIN {X 0,Y 241.933,Z 183.318,A -85,B 0,C 180,E1 -19398.076,E2 -19398.076} C_VEL
LIN {X 0,Y 241.985,Z 183.317,A -85,B 0,C 180,E1 -19402.417,E2 -19402.417} C_VEL
LIN {X 0,Y 241.98,Z 183.299,A -85,B 0,C 180,E1 -19406.507,E2 -19406.507} C_VEL
LIN {X 0,Y 242.036,Z 183.333,A -85,B 0,C 180,E1 -19410.587,E2 -19410.587} C_VEL
LIN {X 0,Y 242.067,Z 183.328,A -85,B 0,C 180,E1 -19414.183,E2 -19414.183} C_VEL
LIN {X 0,Y 242.024,Z 183.32,A -85,B 0,C 180,E1 -19418.313,E2 -19418.313} C_VEL
LIN {X 0,Y 242.162,Z 183.304,A -85,B 0,C 180,E1 -19423.278,E2 -19423.278} C_VEL
LIN {X 0,Y 242.184,Z 183.313,A -85,B 0,C 180,E1 -19428.28,E2 -19428.28} C_VEL
LIN {X 0,Y 242.425,Z 183.266,A -85,B 0,C 180,E1 -19431.665,E2 -19431.665} C_VEL
LIN {X 0,Y 242.252,Z 183.307,A -85,B 0,C 180,E1 -19435.007,E2 -19435.007} C_VEL
LIN {X 0,Y 242.632,Z 183.241,A -85,B 0,C 180,E1 -19438.34,E2 -19438.34} C_VEL
LIN {X 0,Y 242.631,Z 183.261,A -85,B 0,C 180,E1 -19441.66,E2 -19441.66} C_VEL
LIN {X 0,Y 242.412,Z 183.283,A -85,B 0,C 180,E1 -19446.659,E2 -19446.659} C_VEL
LIN {X 0,Y 242.258,Z 183.296,A -85,B 0,C 180,E1 -19450.024,E2 -19450.024} C_VEL
LIN {X 0,Y 242.167,Z 183.299,A -85,B 0,C 180,E1 -19451.185,E2 -19451.185} C_VEL
LIN {X 0,Y 241.462,Z 183.393,A -85,B 0,C 180,E1 -19452.574,E2 -19452.574} C_VEL
LIN {X 0,Y 238.564,Z 183.769,A -85,B 0,C 180,E1 -19454.836,E2 -19454.836} C_VEL
LIN {X 0,Y 236.118,Z 184.061,A -85,B 0,C 180,E1 -19456.68,E2 -19456.68} C_VEL
LIN {X 0,Y 235.069,Z 184.184,A -85,B 0,C 180,E1 -19458.112,E2 -19458.112} C_VEL
LIN {X 0,Y 234.983,Z 184.197,A -85,B 0,C 180,E1 -19458.598,E2 -19458.598} C_VEL
LIN {X 0,Y 234.95,Z 184.205,A -85,B 0,C 180,E1 -19462.884,E2 -19462.884} C_VEL
LIN {X 0,Y 234.966,Z 184.217,A -85,B 0,C 180,E1 -19466.658,E2 -19466.658} C_VEL
LIN {X 0,Y 234.921,Z 184.214,A -85,B 0,C 180,E1 -19470.569,E2 -19470.569} C_VEL
LIN {X 0,Y 234.926,Z 184.186,A -85,B 0,C 180,E1 -19474.639,E2 -19474.639} C_VEL
LIN {X 0,Y 234.941,Z 184.193,A -85,B 0,C 180,E1 -19478.945,E2 -19478.945} C_VEL
LIN {X 0,Y 234.878,Z 184.215,A -85,B 0,C 180,E1 -19483.488,E2 -19483.488} C_VEL
LIN {X 0,Y 234.878,Z 184.219,A -85,B 0,C 180,E1 -19486.512,E2 -19486.512} C_VEL
LIN {X 0,Y 234.928,Z 184.304,A -85,B 0,C 180,E1 -19490.668,E2 -19490.668} C_VEL
LIN {X 0,Y 236.783,Z 191.397,A -85,B 0,C 180,E1 -19494.27,E2 -19494.27} C_VEL
LIN {X 0,Y 237.045,Z 192.421,A -85,B 0,C 180,E1 -19494.619,E2 -19494.619} C_VEL
LIN {X 0,Y 241.553,Z 201.579,A -85,B 0,C 180,E1 -19495.745,E2 -19495.745} C_VEL
LIN {X 0,Y 248.641,Z 217.011,A -85,B 0,C 180,E1 -19497.368,E2 -19497.368} C_VEL
LIN {X 0,Y 252.725,Z 227.313,A -85,B 0,C 180,E1 -19498.295,E2 -19498.295} C_VEL
LIN {X 0,Y 254.73,Z 240.01,A -85,B 0,C 180,E1 -19498.983,E2 -19498.983} C_VEL
LIN {X 0,Y 252.517,Z 300.435,A -85,B 0,C 180,E1 -19500.681,E2 -19500.681} C_VEL
LIN {X 0,Y 251.258,Z 314.314,A -85,B 0,C 180,E1 -19501.379,E2 -19501.379} C_VEL
LIN {X 0,Y 249.552,Z 326.732,A -85,B 0,C 180,E1 -19502.31,E2 -19502.31} C_VEL
LIN {X 0,Y 247.816,Z 337.814,A -85,B 0,C 180,E1 -19503.47,E2 -19503.47} C_VEL
LIN {X 0,Y 245.496,Z 349.362,A -85,B 0,C 180,E1 -19505.023,E2 -19505.023} C_VEL
LIN {X 0,Y 243.124,Z 359.76,A -85,B 0,C 180,E1 -19506.805,E2 -19506.805} C_VEL
LIN {X 0,Y 241.01,Z 368.611,A -85,B 0,C 180,E1 -19508.712,E2 -19508.712} C_VEL
LIN {X 0,Y 238.781,Z 377.471,A -85,B 0,C 180,E1 -19511.109,E2 -19511.109} C_VEL
LIN {X 0,Y 236.815,Z 384.874,A -85,B 0,C 180,E1 -19513.624,E2 -19513.624} C_VEL
LIN {X 0,Y 235.175,Z 390.816,A -85,B 0,C 180,E1 -19516.168,E2 -19516.168} C_VEL
LIN {X 0,Y 234.03,Z 395.511,A -85,B 0,C 180,E1 -19518.743,E2 -19518.743} C_VEL
LIN {X 0,Y 233.284,Z 399.097,A -85,B 0,C 180,E1 -19521.336,E2 -19521.336} C_VEL
LIN {X 0,Y 232.977,Z 400.945,A -85,B 0,C 180,E1 -19523.069,E2 -19523.069} C_VEL
LIN {X 0,Y 232.713,Z 402.643,A -85,B 0,C 180,E1 -19525.283,E2 -19525.283} C_VEL
LIN {X 0,Y 232.67,Z 403.922,A -85,B 0,C 180,E1 -19528.268,E2 -19528.268} C_VEL
LIN {X 0,Y 232.718,Z 404.133,A -85,B 0,C 180,E1 -19529.999,E2 -19529.999} C_VEL
LIN {X 0,Y 232.671,Z 403.911,A -85,B 0,C 180,E1 -19531.73,E2 -19531.73} C_VEL
LIN {X 0,Y 232.768,Z 402.306,A -85,B 0,C 180,E1 -19535.196,E2 -19535.196} C_VEL
LIN {X 0,Y 232.978,Z 400.91,A -85,B 0,C 180,E1 -19536.929,E2 -19536.929} C_VEL
LIN {X 0,Y 233.506,Z 397.98,A -85,B 0,C 180,E1 -19539.527,E2 -19539.527} C_VEL
LIN {X 0,Y 234.377,Z 394.014,A -85,B 0,C 180,E1 -19542.115,E2 -19542.115} C_VEL
LIN {X 0,Y 235.901,Z 387.914,A -85,B 0,C 180,E1 -19545.109,E2 -19545.109} C_VEL
LIN {X 0,Y 237.814,Z 381.253,A -85,B 0,C 180,E1 -19547.631,E2 -19547.631} C_VEL
LIN {X 0,Y 239.956,Z 373.026,A -85,B 0,C 180,E1 -19550.116,E2 -19550.116} C_VEL
LIN {X 0,Y 241.919,Z 364.502,A -85,B 0,C 180,E1 -19552.188,E2 -19552.188} C_VEL
LIN {X 0,Y 244.389,Z 354.02,A -85,B 0,C 180,E1 -19554.19,E2 -19554.19} C_VEL
LIN {X 0,Y 246.85,Z 342.216,A -85,B 0,C 180,E1 -19555.958,E2 -19555.958} C_VEL
LIN {X 0,Y 248.98,Z 330.32,A -85,B 0,C 180,E1 -19557.301,E2 -19557.301} C_VEL
LIN {X 0,Y 250.685,Z 317.933,A -85,B 0,C 180,E1 -19558.348,E2 -19558.348} C_VEL
LIN {X 0,Y 252.081,Z 305.163,A -85,B 0,C 180,E1 -19559.087,E2 -19559.087} C_VEL
LIN {X 0,Y 252.834,Z 291.631,A -85,B 0,C 180,E1 -19559.562,E2 -19559.562} C_VEL
LIN {X 0,Y 254.633,Z 240.043,A -85,B 0,C 180,E1 -19560.981,E2 -19560.981} C_VEL
LIN {X 0,Y 252.474,Z 226.782,A -85,B 0,C 180,E1 -19561.707,E2 -19561.707} C_VEL
LIN {X 0,Y 246.851,Z 213.008,A -85,B 0,C 180,E1 -19562.981,E2 -19562.981} C_VEL
LIN {X 0,Y 240.165,Z 198.888,A -85,B 0,C 180,E1 -19564.519,E2 -19564.519} C_VEL
LIN {X 0,Y 236.998,Z 192.193,A -85,B 0,C 180,E1 -19565.365,E2 -19565.365} C_VEL
LIN {X 0,Y 234.999,Z 184.749,A -85,B 0,C 180,E1 -19568.961,E2 -19568.961} C_VEL
LIN {X 0,Y 234.917,Z 184.214,A -85,B 0,C 180,E1 -19569.471,E2 -19569.471} C_VEL
LIN {X 0,Y 234.88,Z 184.224,A -85,B 0,C 180,E1 -19574.1,E2 -19574.1} C_VEL
LIN {X 0,Y 234.877,Z 184.228,A -85,B 0,C 180,E1 -19578.831,E2 -19578.831} C_VEL
LIN {X 0,Y 234.912,Z 184.194,A -85,B 0,C 180,E1 -19581.077,E2 -19581.077} C_VEL
LIN {X 0,Y 234.921,Z 184.189,A -85,B 0,C 180,E1 -19585.36,E2 -19585.36} C_VEL
LIN {X 0,Y 234.916,Z 184.213,A -85,B 0,C 180,E1 -19589.43,E2 -19589.43} C_VEL
LIN {X 0,Y 234.987,Z 184.213,A -85,B 0,C 180,E1 -19593.793,E2 -19593.793} C_VEL
LIN {X 0,Y 234.984,Z 184.216,A -85,B 0,C 180,E1 -19598.967,E2 -19598.967} C_VEL
LIN {X 0,Y 235.056,Z 184.189,A -85,B 0,C 180,E1 -19603.085,E2 -19603.085} C_VEL
LIN {X 0,Y 235.106,Z 184.179,A -85,B 0,C 180,E1 -19607.922,E2 -19607.922} C_VEL
LIN {X 0,Y 235.367,Z 184.166,A -85,B 0,C 180,E1 -19611.414,E2 -19611.414} C_VEL
LIN {X 0,Y 235.393,Z 184.158,A -85,B 0,C 180,E1 -19613.141,E2 -19613.141} C_VEL
LIN {X 0,Y 235.586,Z 184.138,A -85,B 0,C 180,E1 -19618.291,E2 -19618.291} C_VEL
LIN {X 0,Y 235.586,Z 184.118,A -85,B 0,C 180,E1 -19621.71,E2 -19621.71} C_VEL
LIN {X 0,Y 235.395,Z 184.157,A -85,B 0,C 180,E1 -19626.859,E2 -19626.859} C_VEL
LIN {X 0,Y 235.23,Z 184.164,A -85,B 0,C 180,E1 -19630.327,E2 -19630.327} C_VEL
LIN {X 0,Y 235.104,Z 184.178,A -85,B 0,C 180,E1 -19635.607,E2 -19635.607} C_VEL
LIN {X 0,Y 235.001,Z 184.212,A -85,B 0,C 180,E1 -19639.206,E2 -19639.206} C_VEL
LIN {X 0,Y 234.954,Z 184.203,A -85,B 0,C 180,E1 -19642.884,E2 -19642.884} C_VEL
LIN {X 0,Y 234.963,Z 184.207,A -85,B 0,C 180,E1 -19646.658,E2 -19646.658} C_VEL
LIN {X 0,Y 234.926,Z 184.222,A -85,B 0,C 180,E1 -19650.569,E2 -19650.569} C_VEL
LIN {X 0,Y 234.921,Z 184.168,A -85,B 0,C 180,E1 -19654.64,E2 -19654.64} C_VEL
LIN {X 0,Y 234.937,Z 184.217,A -85,B 0,C 180,E1 -19658.946,E2 -19658.946} C_VEL
LIN {X 0,Y 234.875,Z 184.188,A -85,B 0,C 180,E1 -19663.489,E2 -19663.489} C_VEL
LIN {X 0,Y 234.881,Z 184.226,A -85,B 0,C 180,E1 -19666.515,E2 -19666.515} C_VEL
LIN {X 0,Y 234.914,Z 184.193,A -85,B 0,C 180,E1 -19671.08,E2 -19671.08} C_VEL
LIN {X 0,Y 235.003,Z 184.493,A -85,B 0,C 180,E1 -19672.461,E2 -19672.461} C_VEL
LIN {X 0,Y 236.142,Z 188.708,A -85,B 0,C 180,E1 -19674.528,E2 -19674.528} C_VEL
LIN {X 0,Y 237.967,Z 192.498,A -85,B 0,C 180,E1 -19675.061,E2 -19675.061} C_VEL
LIN {X 0,Y 245.923,Z 208.497,A -85,B 0,C 180,E1 -19676.899,E2 -19676.899} C_VEL
LIN {X 0,Y 251.19,Z 220.576,A -85,B 0,C 180,E1 -19678.081,E2 -19678.081} C_VEL
LIN {X 0,Y 254.289,Z 229.084,A -85,B 0,C 180,E1 -19678.792,E2 -19678.792} C_VEL
LIN {X 0,Y 254.895,Z 233.595,A -85,B 0,C 180,E1 -19679.021,E2 -19679.021} C_VEL
LIN {X 0,Y 252.605,Z 296.374,A -85,B 0,C 180,E1 -19680.784,E2 -19680.784} C_VEL
LIN {X 0,Y 251.341,Z 309.89,A -85,B 0,C 180,E1 -19681.454,E2 -19681.454} C_VEL
LIN {X 0,Y 249.779,Z 322.891,A -85,B 0,C 180,E1 -19682.453,E2 -19682.453} C_VEL
LIN {X 0,Y 247.783,Z 334.71,A -85,B 0,C 180,E1 -19683.695,E2 -19683.695} C_VEL
LIN {X 0,Y 245.58,Z 346.066,A -85,B 0,C 180,E1 -19685.259,E2 -19685.259} C_VEL
LIN {X 0,Y 243.297,Z 356.301,A -85,B 0,C 180,E1 -19687.049,E2 -19687.049} C_VEL
LIN {X 0,Y 241.079,Z 365.899,A -85,B 0,C 180,E1 -19689.191,E2 -19689.191} C_VEL
LIN {X 0,Y 238.91,Z 374.417,A -85,B 0,C 180,E1 -19691.566,E2 -19691.566} C_VEL
LIN {X 0,Y 236.884,Z 381.607,A -85,B 0,C 180,E1 -19694.073,E2 -19694.073} C_VEL
LIN {X 0,Y 235.596,Z 386.455,A -85,B 0,C 180,E1 -19696.195,E2 -19696.195} C_VEL
LIN {X 0,Y 234.366,Z 391.167,A -85,B 0,C 180,E1 -19698.761,E2 -19698.761} C_VEL
LIN {X 0,Y 233.518,Z 394.773,A -85,B 0,C 180,E1 -19701.346,E2 -19701.346} C_VEL
LIN {X 0,Y 233.164,Z 396.635,A -85,B 0,C 180,E1 -19703.076,E2 -19703.076} C_VEL
LIN {X 0,Y 232.921,Z 398.036,A -85,B 0,C 180,E1 -19704.807,E2 -19704.807} C_VEL
LIN {X 0,Y 232.699,Z 399.644,A -85,B 0,C 180,E1 -19708.27,E2 -19708.27} C_VEL
LIN {X 0,Y 232.722,Z 399.874,A -85,B 0,C 180,E1 -19710.001,E2 -19710.001} C_VEL
LIN {X 0,Y 232.698,Z 399.68,A -85,B 0,C 180,E1 -19711.731,E2 -19711.731} C_VEL
LIN {X 0,Y 232.902,Z 398.118,A -85,B 0,C 180,E1 -19715.195,E2 -19715.195} C_VEL
LIN {X 0,Y 233.136,Z 396.753,A -85,B 0,C 180,E1 -19716.926,E2 -19716.926} C_VEL
LIN {X 0,Y 233.779,Z 393.87,A -85,B 0,C 180,E1 -19719.518,E2 -19719.518} C_VEL
LIN {X 0,Y 234.708,Z 389.962,A -85,B 0,C 180,E1 -19722.1,E2 -19722.1} C_VEL
LIN {X 0,Y 236.011,Z 384.923,A -85,B 0,C 180,E1 -19724.662,E2 -19724.662} C_VEL
LIN {X 0,Y 237.773,Z 378.577,A -85,B 0,C 180,E1 -19727.192,E2 -19727.192} C_VEL
LIN {X 0,Y 239.883,Z 370.639,A -85,B 0,C 180,E1 -19729.69,E2 -19729.69} C_VEL
LIN {X 0,Y 242.302,Z 360.769,A -85,B 0,C 180,E1 -19732.152,E2 -19732.152} C_VEL
LIN {X 0,Y 244.67,Z 350.406,A -85,B 0,C 180,E1 -19734.162,E2 -19734.162} C_VEL
LIN {X 0,Y 246.937,Z 340.143,A -85,B 0,C 180,E1 -19735.723,E2 -19735.723} C_VEL
LIN {X 0,Y 248.888,Z 328.913,A -85,B 0,C 180,E1 -19737.086,E2 -19737.086} C_VEL
LIN {X 0,Y 250.713,Z 316.239,A -85,B 0,C 180,E1 -19738.232,E2 -19738.232} C_VEL
LIN {X 0,Y 252.066,Z 303.523,A -85,B 0,C 180,E1 -19739.033,E2 -19739.033} C_VEL
LIN {X 0,Y 252.917,Z 290.389,A -85,B 0,C 180,E1 -19739.553,E2 -19739.553} C_VEL
LIN {X 0,Y 254.963,Z 233.058,A -85,B 0,C 180,E1 -19741.126,E2 -19741.126} C_VEL
LIN {X 0,Y 253.993,Z 227.765,A -85,B 0,C 180,E1 -19741.43,E2 -19741.43} C_VEL
LIN {X 0,Y 247.617,Z 212.119,A -85,B 0,C 180,E1 -19742.865,E2 -19742.865} C_VEL
LIN {X 0,Y 241.484,Z 199.32,A -85,B 0,C 180,E1 -19744.262,E2 -19744.262} C_VEL
LIN {X 0,Y 236.193,Z 188.911,A -85,B 0,C 180,E1 -19745.577,E2 -19745.577} C_VEL
LIN {X 0,Y 235.231,Z 185.355,A -85,B 0,C 180,E1 -19747.229,E2 -19747.229} C_VEL
LIN {X 0,Y 234.983,Z 184.239,A -85,B 0,C 180,E1 -19747.951,E2 -19747.951} C_VEL
LIN {X 0,Y 234.877,Z 184.204,A -85,B 0,C 180,E1 -19751.578,E2 -19751.578} C_VEL
LIN {X 0,Y 234.887,Z 184.19,A -85,B 0,C 180,E1 -19755.897,E2 -19755.897} C_VEL
LIN {X 0,Y 234.881,Z 184.207,A -85,B 0,C 180,E1 -19758.831,E2 -19758.831} C_VEL
LIN {X 0,Y 234.918,Z 184.222,A -85,B 0,C 180,E1 -19761.078,E2 -19761.078} C_VEL
LIN {X 0,Y 234.926,Z 184.166,A -85,B 0,C 180,E1 -19765.361,E2 -19765.361} C_VEL
LIN {X 0,Y 234.931,Z 184.221,A -85,B 0,C 180,E1 -19769.432,E2 -19769.432} C_VEL
LIN {X 0,Y 234.993,Z 184.205,A -85,B 0,C 180,E1 -19773.794,E2 -19773.794} C_VEL
LIN {X 0,Y 234.996,Z 184.198,A -85,B 0,C 180,E1 -19778.968,E2 -19778.968} C_VEL
LIN {X 0,Y 235.094,Z 184.186,A -85,B 0,C 180,E1 -19783.06,E2 -19783.06} C_VEL
LIN {X 0,Y 235.144,Z 184.192,A -85,B 0,C 180,E1 -19787.923,E2 -19787.923} C_VEL
LIN {X 0,Y 235.375,Z 184.142,A -85,B 0,C 180,E1 -19791.414,E2 -19791.414} C_VEL
LIN {X 0,Y 235.401,Z 184.156,A -85,B 0,C 180,E1 -19793.141,E2 -19793.141} C_VEL
LIN {X 0,Y 235.591,Z 184.117,A -85,B 0,C 180,E1 -19798.29,E2 -19798.29} C_VEL
LIN {X 0,Y 235.591,Z 184.138,A -85,B 0,C 180,E1 -19801.709,E2 -19801.709} C_VEL
LIN {X 0,Y 235.362,Z 184.162,A -85,B 0,C 180,E1 -19806.86,E2 -19806.86} C_VEL
LIN {X 0,Y 235.183,Z 184.173,A -85,B 0,C 180,E1 -19810.329,E2 -19810.329} C_VEL
LIN {X 0,Y 235.083,Z 184.198,A -85,B 0,C 180,E1 -19815.608,E2 -19815.608} C_VEL
LIN {X 0,Y 234.983,Z 184.197,A -85,B 0,C 180,E1 -19818.598,E2 -19818.598} C_VEL
LIN {X 0,Y 234.305,Z 184.296,A -85,B 0,C 180,E1 -19820.029,E2 -19820.029} C_VEL
LIN {X 0,Y 231.431,Z 184.649,A -85,B 0,C 180,E1 -19822.363,E2 -19822.363} C_VEL
LIN {X 0,Y 229.008,Z 184.949,A -85,B 0,C 180,E1 -19824.266,E2 -19824.266} C_VEL
LIN {X 0,Y 227.995,Z 185.08,A -85,B 0,C 180,E1 -19825.744,E2 -19825.744} C_VEL
LIN {X 0,Y 227.926,Z 185.091,A -85,B 0,C 180,E1 -19826.245,E2 -19826.245} C_VEL
LIN {X 0,Y 227.896,Z 185.086,A -85,B 0,C 180,E1 -19830.291,E2 -19830.291} C_VEL
LIN {X 0,Y 227.876,Z 185.081,A -85,B 0,C 180,E1 -19833.721,E2 -19833.721} C_VEL
LIN {X 0,Y 227.842,Z 185.061,A -85,B 0,C 180,E1 -19838.091,E2 -19838.091} C_VEL
LIN {X 0,Y 227.805,Z 185.095,A -85,B 0,C 180,E1 -19842.744,E2 -19842.744} C_VEL
LIN {X 0,Y 227.806,Z 185.099,A -85,B 0,C 180,E1 -19847.257,E2 -19847.257} C_VEL
LIN {X 0,Y 227.906,Z 185.276,A -85,B 0,C 180,E1 -19849.758,E2 -19849.758} C_VEL
LIN {X 0,Y 229.766,Z 192.122,A -85,B 0,C 180,E1 -19853.286,E2 -19853.286} C_VEL
LIN {X 0,Y 233.141,Z 199.006,A -85,B 0,C 180,E1 -19854.232,E2 -19854.232} C_VEL
LIN {X 0,Y 238.24,Z 209.335,A -85,B 0,C 180,E1 -19855.48,E2 -19855.48} C_VEL
LIN {X 0,Y 244.6,Z 223.866,A -85,B 0,C 180,E1 -19856.996,E2 -19856.996} C_VEL
LIN {X 0,Y 247.049,Z 230.562,A -85,B 0,C 180,E1 -19857.59,E2 -19857.59} C_VEL
LIN {X 0,Y 248.651,Z 241.262,A -85,B 0,C 180,E1 -19858.18,E2 -19858.18} C_VEL
LIN {X 0,Y 246.371,Z 300.397,A -85,B 0,C 180,E1 -19859.876,E2 -19859.876} C_VEL
LIN {X 0,Y 245.06,Z 314.26,A -85,B 0,C 180,E1 -19860.586,E2 -19860.586} C_VEL
LIN {X 0,Y 243.296,Z 326.674,A -85,B 0,C 180,E1 -19861.534,E2 -19861.534} C_VEL
LIN {X 0,Y 241.468,Z 337.754,A -85,B 0,C 180,E1 -19862.716,E2 -19862.716} C_VEL
LIN {X 0,Y 239.066,Z 349.301,A -85,B 0,C 180,E1 -19864.303,E2 -19864.303} C_VEL
LIN {X 0,Y 236.611,Z 359.698,A -85,B 0,C 180,E1 -19866.127,E2 -19866.127} C_VEL
LIN {X 0,Y 234.486,Z 368.201,A -85,B 0,C 180,E1 -19867.998,E2 -19867.998} C_VEL
LIN {X 0,Y 232.433,Z 376.209,A -85,B 0,C 180,E1 -19870.168,E2 -19870.168} C_VEL
LIN {X 0,Y 230.321,Z 383.693,A -85,B 0,C 180,E1 -19872.692,E2 -19872.692} C_VEL
LIN {X 0,Y 228.254,Z 390.752,A -85,B 0,C 180,E1 -19875.74,E2 -19875.74} C_VEL
LIN {X 0,Y 227.053,Z 395.447,A -85,B 0,C 180,E1 -19878.393,E2 -19878.393} C_VEL
LIN {X 0,Y 226.257,Z 399.032,A -85,B 0,C 180,E1 -19881.065,E2 -19881.065} C_VEL
LIN {X 0,Y 225.918,Z 400.88,A -85,B 0,C 180,E1 -19882.851,E2 -19882.851} C_VEL
LIN {X 0,Y 225.61,Z 402.772,A -85,B 0,C 180,E1 -19885.441,E2 -19885.441} C_VEL
LIN {X 0,Y 225.57,Z 403.857,A -85,B 0,C 180,E1 -19888.214,E2 -19888.214} C_VEL
LIN {X 0,Y 225.635,Z 404.068,A -85,B 0,C 180,E1 -19889.999,E2 -19889.999} C_VEL
LIN {X 0,Y 225.571,Z 403.846,A -85,B 0,C 180,E1 -19891.785,E2 -19891.785} C_VEL
LIN {X 0,Y 225.692,Z 402.241,A -85,B 0,C 180,E1 -19895.359,E2 -19895.359} C_VEL
LIN {X 0,Y 225.919,Z 400.845,A -85,B 0,C 180,E1 -19897.147,E2 -19897.147} C_VEL
LIN {X 0,Y 226.49,Z 397.914,A -85,B 0,C 180,E1 -19899.825,E2 -19899.825} C_VEL
LIN {X 0,Y 227.428,Z 393.948,A -85,B 0,C 180,E1 -19902.492,E2 -19902.492} C_VEL
LIN {X 0,Y 229.044,Z 387.848,A -85,B 0,C 180,E1 -19905.573,E2 -19905.573} C_VEL
LIN {X 0,Y 231.029,Z 381.186,A -85,B 0,C 180,E1 -19908.167,E2 -19908.167} C_VEL
LIN {X 0,Y 233.306,Z 372.803,A -85,B 0,C 180,E1 -19910.764,E2 -19910.764} C_VEL
LIN {X 0,Y 235.356,Z 364.434,A -85,B 0,C 180,E1 -19912.841,E2 -19912.841} C_VEL
LIN {X 0,Y 237.923,Z 353.951,A -85,B 0,C 180,E1 -19914.892,E2 -19914.892} C_VEL
LIN {X 0,Y 240.481,Z 342.147,A -85,B 0,C 180,E1 -19916.699,E2 -19916.699} C_VEL
LIN {X 0,Y 242.695,Z 330.249,A -85,B 0,C 180,E1 -19918.07,E2 -19918.07} C_VEL
LIN {X 0,Y 244.474,Z 317.86,A -85,B 0,C 180,E1 -19919.136,E2 -19919.136} C_VEL
LIN {X 0,Y 245.886,Z 305.413,A -85,B 0,C 180,E1 -19919.873,E2 -19919.873} C_VEL
LIN {X 0,Y 246.717,Z 290.842,A -85,B 0,C 180,E1 -19920.395,E2 -19920.395} C_VEL
LIN {X 0,Y 248.514,Z 240.722,A -85,B 0,C 180,E1 -19921.806,E2 -19921.806} C_VEL
LIN {X 0,Y 246.601,Z 229.188,A -85,B 0,C 180,E1 -19922.47,E2 -19922.47} C_VEL
LIN {X 0,Y 240.674,Z 214.666,A -85,B 0,C 180,E1 -19923.879,E2 -19923.879} C_VEL
LIN {X 0,Y 233.46,Z 199.564,A -85,B 0,C 180,E1 -19925.629,E2 -19925.629} C_VEL
LIN {X 0,Y 229.715,Z 192.14,A -85,B 0,C 180,E1 -19926.656,E2 -19926.656} C_VEL
LIN {X 0,Y 227.932,Z 185.347,A -85,B 0,C 180,E1 -19930.111,E2 -19930.111} C_VEL
LIN {X 0,Y 227.874,Z 185.115,A -85,B 0,C 180,E1 -19930.364,E2 -19930.364} C_VEL
LIN {X 0,Y 227.821,Z 185.105,A -85,B 0,C 180,E1 -19935.194,E2 -19935.194} C_VEL
LIN {X 0,Y 227.82,Z 185.106,A -85,B 0,C 180,E1 -19939.622,E2 -19939.622} C_VEL
LIN {X 0,Y 227.874,Z 185.05,A -85,B 0,C 180,E1 -19944.127,E2 -19944.127} C_VEL
LIN {X 0,Y 227.86,Z 185.102,A -85,B 0,C 180,E1 -19948.376,E2 -19948.376} C_VEL
LIN {X 0,Y 227.872,Z 185.098,A -85,B 0,C 180,E1 -19952.443,E2 -19952.443} C_VEL
LIN {X 0,Y 227.899,Z 185.079,A -85,B 0,C 180,E1 -19956.366,E2 -19956.366} C_VEL
LIN {X 0,Y 227.919,Z 185.088,A -85,B 0,C 180,E1 -19960.172,E2 -19960.172} C_VEL
LIN {X 0,Y 228.022,Z 185.075,A -85,B 0,C 180,E1 -19963.895,E2 -19963.895} C_VEL
LIN {X 0,Y 228.062,Z 185.059,A -85,B 0,C 180,E1 -19967.543,E2 -19967.543} C_VEL
LIN {X 0,Y 228.297,Z 185.045,A -85,B 0,C 180,E1 -19971.146,E2 -19971.146} C_VEL
LIN {X 0,Y 228.344,Z 185.037,A -85,B 0,C 180,E1 -19972.928,E2 -19972.928} C_VEL
LIN {X 0,Y 228.544,Z 185.015,A -85,B 0,C 180,E1 -19978.238,E2 -19978.238} C_VEL
LIN {X 0,Y 228.544,Z 184.994,A -85,B 0,C 180,E1 -19981.762,E2 -19981.762} C_VEL
LIN {X 0,Y 228.346,Z 185.035,A -85,B 0,C 180,E1 -19987.072,E2 -19987.072} C_VEL
LIN {X 0,Y 228.156,Z 185.048,A -85,B 0,C 180,E1 -19990.651,E2 -19990.651} C_VEL
LIN {X 0,Y 228.055,Z 185.064,A -85,B 0,C 180,E1 -19994.273,E2 -19994.273} C_VEL
LIN {X 0,Y 227.996,Z 185.08,A -85,B 0,C 180,E1 -19997.954,E2 -19997.954} C_VEL
LIN {X 0,Y 227.923,Z 185.076,A -85,B 0,C 180,E1 -20002.33,E2 -20002.33} C_VEL
LIN {X 0,Y 227.937,Z 185.082,A -85,B 0,C 180,E1 -20006.604,E2 -20006.604} C_VEL
LIN {X 0,Y 227.903,Z 185.098,A -85,B 0,C 180,E1 -20010.297,E2 -20010.297} C_VEL
LIN {X 0,Y 227.871,Z 185.053,A -85,B 0,C 180,E1 -20013.722,E2 -20013.722} C_VEL
LIN {X 0,Y 227.838,Z 185.083,A -85,B 0,C 180,E1 -20018.092,E2 -20018.092} C_VEL
LIN {X 0,Y 227.802,Z 185.07,A -85,B 0,C 180,E1 -20022.745,E2 -20022.745} C_VEL
LIN {X 0,Y 227.804,Z 185.107,A -85,B 0,C 180,E1 -20027.258,E2 -20027.258} C_VEL
LIN {X 0,Y 227.916,Z 185.274,A -85,B 0,C 180,E1 -20031.394,E2 -20031.394} C_VEL
LIN {X 0,Y 228.908,Z 188.892,A -85,B 0,C 180,E1 -20033.249,E2 -20033.249} C_VEL
LIN {X 0,Y 235.229,Z 200.924,A -85,B 0,C 180,E1 -20034.901,E2 -20034.901} C_VEL
LIN {X 0,Y 242.655,Z 216.667,A -85,B 0,C 180,E1 -20036.677,E2 -20036.677} C_VEL
LIN {X 0,Y 248.32,Z 230.947,A -85,B 0,C 180,E1 -20038.014,E2 -20038.014} C_VEL
LIN {X 0,Y 248.826,Z 234.459,A -85,B 0,C 180,E1 -20038.204,E2 -20038.204} C_VEL
LIN {X 0,Y 246.477,Z 296.04,A -85,B 0,C 180,E1 -20039.962,E2 -20039.962} C_VEL
LIN {X 0,Y 245.191,Z 309.324,A -85,B 0,C 180,E1 -20040.619,E2 -20040.619} C_VEL
LIN {X 0,Y 243.688,Z 321.875,A -85,B 0,C 180,E1 -20041.586,E2 -20041.586} C_VEL
LIN {X 0,Y 241.76,Z 333.196,A -85,B 0,C 180,E1 -20042.753,E2 -20042.753} C_VEL
LIN {X 0,Y 239.426,Z 344.846,A -85,B 0,C 180,E1 -20044.346,E2 -20044.346} C_VEL
LIN {X 0,Y 237.01,Z 355.311,A -85,B 0,C 180,E1 -20046.172,E2 -20046.172} C_VEL
LIN {X 0,Y 234.631,Z 365.29,A -85,B 0,C 180,E1 -20048.4,E2 -20048.4} C_VEL
LIN {X 0,Y 232.548,Z 373.132,A -85,B 0,C 180,E1 -20050.584,E2 -20050.584} C_VEL
LIN {X 0,Y 230.341,Z 380.56,A -85,B 0,C 180,E1 -20053.152,E2 -20053.152} C_VEL
LIN {X 0,Y 228.697,Z 386.521,A -85,B 0,C 180,E1 -20055.769,E2 -20055.769} C_VEL
LIN {X 0,Y 227.39,Z 391.233,A -85,B 0,C 180,E1 -20058.412,E2 -20058.412} C_VEL
LIN {X 0,Y 226.502,Z 394.839,A -85,B 0,C 180,E1 -20061.076,E2 -20061.076} C_VEL
LIN {X 0,Y 226.106,Z 396.701,A -85,B 0,C 180,E1 -20062.859,E2 -20062.859} C_VEL
LIN {X 0,Y 225.825,Z 398.202,A -85,B 0,C 180,E1 -20064.806,E2 -20064.806} C_VEL
LIN {X 0,Y 225.601,Z 399.709,A -85,B 0,C 180,E1 -20068.216,E2 -20068.216} C_VEL
LIN {X 0,Y 225.638,Z 399.939,A -85,B 0,C 180,E1 -20070.001,E2 -20070.001} C_VEL
LIN {X 0,Y 225.6,Z 399.745,A -85,B 0,C 180,E1 -20071.786,E2 -20071.786} C_VEL
LIN {X 0,Y 225.844,Z 398.182,A -85,B 0,C 180,E1 -20075.357,E2 -20075.357} C_VEL
LIN {X 0,Y 226.088,Z 396.817,A -85,B 0,C 180,E1 -20077.143,E2 -20077.143} C_VEL
LIN {X 0,Y 226.78,Z 393.934,A -85,B 0,C 180,E1 -20079.814,E2 -20079.814} C_VEL
LIN {X 0,Y 227.753,Z 390.026,A -85,B 0,C 180,E1 -20082.475,E2 -20082.475} C_VEL
LIN {X 0,Y 229.114,Z 384.986,A -85,B 0,C 180,E1 -20085.114,E2 -20085.114} C_VEL
LIN {X 0,Y 230.991,Z 378.64,A -85,B 0,C 180,E1 -20087.714,E2 -20087.714} C_VEL
LIN {X 0,Y 233.181,Z 370.702,A -85,B 0,C 180,E1 -20090.28,E2 -20090.28} C_VEL
LIN {X 0,Y 235.454,Z 361.853,A -85,B 0,C 180,E1 -20092.567,E2 -20092.567} C_VEL
LIN {X 0,Y 237.95,Z 351.639,A -85,B 0,C 180,E1 -20094.657,E2 -20094.657} C_VEL
LIN {X 0,Y 240.566,Z 340.203,A -85,B 0,C 180,E1 -20096.457,E2 -20096.457} C_VEL
LIN {X 0,Y 242.601,Z 328.972,A -85,B 0,C 180,E1 -20097.848,E2 -20097.848} C_VEL
LIN {X 0,Y 244.484,Z 316.295,A -85,B 0,C 180,E1 -20099.019,E2 -20099.019} C_VEL
LIN {X 0,Y 245.988,Z 302.661,A -85,B 0,C 180,E1 -20099.881,E2 -20099.881} C_VEL
LIN {X 0,Y 246.767,Z 290.434,A -85,B 0,C 180,E1 -20100.366,E2 -20100.366} C_VEL
LIN {X 0,Y 248.814,Z 233.061,A -85,B 0,C 180,E1 -20101.986,E2 -20101.986} C_VEL
LIN {X 0,Y 247.849,Z 229.388,A -85,B 0,C 180,E1 -20102.249,E2 -20102.249} C_VEL
LIN {X 0,Y 241.189,Z 213.226,A -85,B 0,C 180,E1 -20103.82,E2 -20103.82} C_VEL
LIN {X 0,Y 234.074,Z 198.737,A -85,B 0,C 180,E1 -20105.531,E2 -20105.531} C_VEL
LIN {X 0,Y 228.942,Z 188.901,A -85,B 0,C 180,E1 -20106.898,E2 -20106.898} C_VEL
LIN {X 0,Y 227.918,Z 185.306,A -85,B 0,C 180,E1 -20108.742,E2 -20108.742} C_VEL
LIN {X 0,Y 227.821,Z 185.072,A -85,B 0,C 180,E1 -20110.378,E2 -20110.378} C_VEL
LIN {X 0,Y 227.829,Z 185.075,A -85,B 0,C 180,E1 -20115.194,E2 -20115.194} C_VEL
LIN {X 0,Y 227.824,Z 185.1,A -85,B 0,C 180,E1 -20119.623,E2 -20119.623} C_VEL
LIN {X 0,Y 227.879,Z 185.045,A -85,B 0,C 180,E1 -20124.128,E2 -20124.128} C_VEL
LIN {X 0,Y 227.87,Z 185.09,A -85,B 0,C 180,E1 -20128.377,E2 -20128.377} C_VEL
LIN {X 0,Y 227.884,Z 185.082,A -85,B 0,C 180,E1 -20132.445,E2 -20132.445} C_VEL
LIN {X 0,Y 227.905,Z 185.09,A -85,B 0,C 180,E1 -20136.366,E2 -20136.366} C_VEL
LIN {X 0,Y 227.935,Z 185.089,A -85,B 0,C 180,E1 -20140.174,E2 -20140.174} C_VEL
LIN {X 0,Y 228.052,Z 185.056,A -85,B 0,C 180,E1 -20143.897,E2 -20143.897} C_VEL
LIN {X 0,Y 228.162,Z 185.048,A -85,B 0,C 180,E1 -20149.349,E2 -20149.349} C_VEL
LIN {X 0,Y 228.352,Z 185.034,A -85,B 0,C 180,E1 -20152.928,E2 -20152.928} C_VEL
LIN {X 0,Y 228.55,Z 184.994,A -85,B 0,C 180,E1 -20158.238,E2 -20158.238} C_VEL
LIN {X 0,Y 228.549,Z 185.014,A -85,B 0,C 180,E1 -20161.762,E2 -20161.762} C_VEL
LIN {X 0,Y 228.313,Z 185.041,A -85,B 0,C 180,E1 -20167.073,E2 -20167.073} C_VEL
LIN {X 0,Y 228.125,Z 185.049,A -85,B 0,C 180,E1 -20170.652,E2 -20170.652} C_VEL
LIN {X 0,Y 228.037,Z 185.079,A -85,B 0,C 180,E1 -20174.274,E2 -20174.274} C_VEL
LIN {X 0,Y 227.927,Z 185.074,A -85,B 0,C 180,E1 -20178.578,E2 -20178.578} C_VEL
LIN {X 0,Y 227.914,Z 185.088,A -85,B 0,C 180,E1 -20182.32,E2 -20182.32} C_VEL
LIN {X 0,Y 227.926,Z 185.091,A -85,B 0,C 180,E1 -20186.245,E2 -20186.245} C_VEL
LIN {X 0,Y 227.628,Z 185.135,A -85,B 0,C 180,E1 -20187.23,E2 -20187.23} C_VEL
LIN {X 0,Y 226.274,Z 185.309,A -85,B 0,C 180,E1 -20188.686,E2 -20188.686} C_VEL
LIN {X 0,Y 221.898,Z 185.845,A -85,B 0,C 180,E1 -20192.083,E2 -20192.083} C_VEL
LIN {X 0,Y 220.871,Z 185.954,A -85,B 0,C 180,E1 -20193.609,E2 -20193.609} C_VEL
LIN {X 0,Y 220.805,Z 185.951,A -85,B 0,C 180,E1 -20194.126,E2 -20194.126} C_VEL
LIN {X 0,Y 220.808,Z 185.929,A -85,B 0,C 180,E1 -20197.278,E2 -20197.278} C_VEL
LIN {X 0,Y 220.794,Z 185.979,A -85,B 0,C 180,E1 -20200.188,E2 -20200.188} C_VEL
LIN {X 0,Y 220.767,Z 185.98,A -85,B 0,C 180,E1 -20204.456,E2 -20204.456} C_VEL
LIN {X 0,Y 220.819,Z 186.15,A -85,B 0,C 180,E1 -20208.673,E2 -20208.673} C_VEL
LIN {X 0,Y 222.377,Z 191.985,A -85,B 0,C 180,E1 -20211.842,E2 -20211.842} C_VEL
LIN {X 0,Y 226.03,Z 198.969,A -85,B 0,C 180,E1 -20212.923,E2 -20212.923} C_VEL
LIN {X 0,Y 231.426,Z 209.604,A -85,B 0,C 180,E1 -20214.323,E2 -20214.323} C_VEL
LIN {X 0,Y 238.445,Z 225.419,A -85,B 0,C 180,E1 -20216.087,E2 -20216.087} C_VEL
LIN {X 0,Y 241.254,Z 232.977,A -85,B 0,C 180,E1 -20216.797,E2 -20216.797} C_VEL
LIN {X 0,Y 242.598,Z 242.828,A -85,B 0,C 180,E1 -20217.344,E2 -20217.344} C_VEL
LIN {X 0,Y 240.301,Z 299.976,A -85,B 0,C 180,E1 -20219.013,E2 -20219.013} C_VEL
LIN {X 0,Y 238.988,Z 313.571,A -85,B 0,C 180,E1 -20219.711,E2 -20219.711} C_VEL
LIN {X 0,Y 237.263,Z 325.509,A -85,B 0,C 180,E1 -20220.62,E2 -20220.62} C_VEL
LIN {X 0,Y 235.178,Z 337.694,A -85,B 0,C 180,E1 -20221.922,E2 -20221.922} C_VEL
LIN {X 0,Y 232.692,Z 349.24,A -85,B 0,C 180,E1 -20223.545,E2 -20223.545} C_VEL
LIN {X 0,Y 230.127,Z 359.637,A -85,B 0,C 180,E1 -20225.411,E2 -20225.411} C_VEL
LIN {X 0,Y 227.888,Z 368.135,A -85,B 0,C 180,E1 -20227.325,E2 -20227.325} C_VEL
LIN {X 0,Y 225.38,Z 377.346,A -85,B 0,C 180,E1 -20229.939,E2 -20229.939} C_VEL
LIN {X 0,Y 223.181,Z 384.747,A -85,B 0,C 180,E1 -20232.593,E2 -20232.593} C_VEL
LIN {X 0,Y 221.345,Z 390.688,A -85,B 0,C 180,E1 -20235.285,E2 -20235.285} C_VEL
LIN {X 0,Y 220.094,Z 395.383,A -85,B 0,C 180,E1 -20238.02,E2 -20238.02} C_VEL
LIN {X 0,Y 219.222,Z 398.968,A -85,B 0,C 180,E1 -20240.775,E2 -20240.775} C_VEL
LIN {X 0,Y 218.854,Z 400.816,A -85,B 0,C 180,E1 -20242.619,E2 -20242.619} C_VEL
LIN {X 0,Y 218.514,Z 402.877,A -85,B 0,C 180,E1 -20245.596,E2 -20245.596} C_VEL
LIN {X 0,Y 218.474,Z 403.792,A -85,B 0,C 180,E1 -20248.156,E2 -20248.156} C_VEL
LIN {X 0,Y 218.534,Z 404.003,A -85,B 0,C 180,E1 -20249.999,E2 -20249.999} C_VEL
LIN {X 0,Y 218.474,Z 403.781,A -85,B 0,C 180,E1 -20251.843,E2 -20251.843} C_VEL
LIN {X 0,Y 218.513,Z 402.856,A -85,B 0,C 180,E1 -20254.402,E2 -20254.402} C_VEL
LIN {X 0,Y 218.855,Z 400.779,A -85,B 0,C 180,E1 -20257.379,E2 -20257.379} C_VEL
LIN {X 0,Y 219.492,Z 397.848,A -85,B 0,C 180,E1 -20260.142,E2 -20260.142} C_VEL
LIN {X 0,Y 220.49,Z 393.882,A -85,B 0,C 180,E1 -20262.891,E2 -20262.891} C_VEL
LIN {X 0,Y 222.201,Z 387.781,A -85,B 0,C 180,E1 -20266.065,E2 -20266.065} C_VEL
LIN {X 0,Y 224.267,Z 381.119,A -85,B 0,C 180,E1 -20268.735,E2 -20268.735} C_VEL
LIN {X 0,Y 226.519,Z 373.27,A -85,B 0,C 180,E1 -20271.244,E2 -20271.244} C_VEL
LIN {X 0,Y 228.804,Z 364.366,A -85,B 0,C 180,E1 -20273.534,E2 -20273.534} C_VEL
LIN {X 0,Y 231.505,Z 353.883,A -85,B 0,C 180,E1 -20275.631,E2 -20275.631} C_VEL
LIN {X 0,Y 234.166,Z 342.078,A -85,B 0,C 180,E1 -20277.479,E2 -20277.479} C_VEL
LIN {X 0,Y 236.466,Z 330.178,A -85,B 0,C 180,E1 -20278.878,E2 -20278.878} C_VEL
LIN {X 0,Y 238.304,Z 317.788,A -85,B 0,C 180,E1 -20279.966,E2 -20279.966} C_VEL
LIN {X 0,Y 239.814,Z 304.881,A -85,B 0,C 180,E1 -20280.738,E2 -20280.738} C_VEL
LIN {X 0,Y 240.636,Z 290.584,A -85,B 0,C 180,E1 -20281.254,E2 -20281.254} C_VEL
LIN {X 0,Y 242.458,Z 241.496,A -85,B 0,C 180,E1 -20282.668,E2 -20282.668} C_VEL
LIN {X 0,Y 240.906,Z 231.929,A -85,B 0,C 180,E1 -20283.238,E2 -20283.238} C_VEL
LIN {X 0,Y 235.409,Z 218.336,A -85,B 0,C 180,E1 -20284.608,E2 -20284.608} C_VEL
LIN {X 0,Y 228.107,Z 202.962,A -85,B 0,C 180,E1 -20286.466,E2 -20286.466} C_VEL
LIN {X 0,Y 223.929,Z 195.18,A -85,B 0,C 180,E1 -20287.565,E2 -20287.565} C_VEL
LIN {X 0,Y 222.403,Z 191.964,A -85,B 0,C 180,E1 -20288.099,E2 -20288.099} C_VEL
LIN {X 0,Y 220.828,Z 186.259,A -85,B 0,C 180,E1 -20291.17,E2 -20291.17} C_VEL
LIN {X 0,Y 220.769,Z 185.979,A -85,B 0,C 180,E1 -20291.951,E2 -20291.951} C_VEL
LIN {X 0,Y 220.763,Z 185.979,A -85,B 0,C 180,E1 -20295.543,E2 -20295.543} C_VEL
LIN {X 0,Y 220.801,Z 185.962,A -85,B 0,C 180,E1 -20300.462,E2 -20300.462} C_VEL
LIN {X 0,Y 220.795,Z 185.94,A -85,B 0,C 180,E1 -20305.044,E2 -20305.044} C_VEL
LIN {X 0,Y 220.828,Z 185.968,A -85,B 0,C 180,E1 -20309.389,E2 -20309.389} C_VEL
LIN {X 0,Y 220.887,Z 185.97,A -85,B 0,C 180,E1 -20313.548,E2 -20313.548} C_VEL
LIN {X 0,Y 220.857,Z 185.965,A -85,B 0,C 180,E1 -20317.551,E2 -20317.551} C_VEL
LIN {X 0,Y 220.955,Z 185.942,A -85,B 0,C 180,E1 -20322.589,E2 -20322.589} C_VEL
LIN {X 0,Y 220.998,Z 185.942,A -85,B 0,C 180,E1 -20327.138,E2 -20327.138} C_VEL
LIN {X 0,Y 221.228,Z 185.922,A -85,B 0,C 180,E1 -20330.86,E2 -20330.86} C_VEL
LIN {X 0,Y 221.28,Z 185.918,A -85,B 0,C 180,E1 -20332.701,E2 -20332.701} C_VEL
LIN {X 0,Y 221.502,Z 185.892,A -85,B 0,C 180,E1 -20338.182,E2 -20338.182} C_VEL
LIN {X 0,Y 221.502,Z 185.871,A -85,B 0,C 180,E1 -20341.818,E2 -20341.818} C_VEL
LIN {X 0,Y 221.281,Z 185.911,A -85,B 0,C 180,E1 -20347.299,E2 -20347.299} C_VEL
LIN {X 0,Y 221.105,Z 185.93,A -85,B 0,C 180,E1 -20350.995,E2 -20350.995} C_VEL
LIN {X 0,Y 221.009,Z 185.935,A -85,B 0,C 180,E1 -20356.631,E2 -20356.631} C_VEL
LIN {X 0,Y 220.886,Z 185.962,A -85,B 0,C 180,E1 -20360.487,E2 -20360.487} C_VEL
LIN {X 0,Y 220.861,Z 185.972,A -85,B 0,C 180,E1 -20364.436,E2 -20364.436} C_VEL
LIN {X 0,Y 220.831,Z 185.963,A -85,B 0,C 180,E1 -20368.515,E2 -20368.515} C_VEL
LIN {X 0,Y 220.812,Z 185.947,A -85,B 0,C 180,E1 -20372.757,E2 -20372.757} C_VEL
LIN {X 0,Y 220.804,Z 185.941,A -85,B 0,C 180,E1 -20377.279,E2 -20377.279} C_VEL
LIN {X 0,Y 220.789,Z 185.981,A -85,B 0,C 180,E1 -20380.189,E2 -20380.189} C_VEL
LIN {X 0,Y 220.766,Z 185.948,A -85,B 0,C 180,E1 -20384.456,E2 -20384.456} C_VEL
LIN {X 0,Y 220.761,Z 185.968,A -85,B 0,C 180,E1 -20388.048,E2 -20388.048} C_VEL
LIN {X 0,Y 220.821,Z 186.125,A -85,B 0,C 180,E1 -20390.309,E2 -20390.309} C_VEL
LIN {X 0,Y 221.622,Z 189.024,A -85,B 0,C 180,E1 -20391.836,E2 -20391.836} C_VEL
LIN {X 0,Y 226.606,Z 198.123,A -85,B 0,C 180,E1 -20393.241,E2 -20393.241} C_VEL
LIN {X 0,Y 233.703,Z 212.165,A -85,B 0,C 180,E1 -20395.051,E2 -20395.051} C_VEL
LIN {X 0,Y 239.919,Z 226.445,A -85,B 0,C 180,E1 -20396.589,E2 -20396.589} C_VEL
LIN {X 0,Y 242.75,Z 234.488,A -85,B 0,C 180,E1 -20397.308,E2 -20397.308} C_VEL
LIN {X 0,Y 240.307,Z 296.794,A -85,B 0,C 180,E1 -20399.144,E2 -20399.144} C_VEL
LIN {X 0,Y 238.956,Z 310.184,A -85,B 0,C 180,E1 -20399.837,E2 -20399.837} C_VEL
LIN {X 0,Y 237.29,Z 323.035,A -85,B 0,C 180,E1 -20400.868,E2 -20400.868} C_VEL
LIN {X 0,Y 235.16,Z 334.851,A -85,B 0,C 180,E1 -20402.164,E2 -20402.164} C_VEL
LIN {X 0,Y 232.758,Z 346.205,A -85,B 0,C 180,E1 -20403.796,E2 -20403.796} C_VEL
LIN {X 0,Y 230.268,Z 356.438,A -85,B 0,C 180,E1 -20405.669,E2 -20405.669} C_VEL
LIN {X 0,Y 227.882,Z 365.918,A -85,B 0,C 180,E1 -20407.891,E2 -20407.891} C_VEL
LIN {X 0,Y 225.471,Z 374.551,A -85,B 0,C 180,E1 -20410.424,E2 -20410.424} C_VEL
LIN {X 0,Y 223.206,Z 381.741,A -85,B 0,C 180,E1 -20413.068,E2 -20413.068} C_VEL
LIN {X 0,Y 221.789,Z 386.588,A -85,B 0,C 180,E1 -20415.316,E2 -20415.316} C_VEL
LIN {X 0,Y 220.412,Z 391.299,A -85,B 0,C 180,E1 -20418.039,E2 -20418.039} C_VEL
LIN {X 0,Y 219.481,Z 394.905,A -85,B 0,C 180,E1 -20420.788,E2 -20420.788} C_VEL
LIN {X 0,Y 219.053,Z 396.767,A -85,B 0,C 180,E1 -20422.628,E2 -20422.628} C_VEL
LIN {X 0,Y 218.69,Z 398.509,A -85,B 0,C 180,E1 -20425.034,E2 -20425.034} C_VEL
LIN {X 0,Y 218.506,Z 399.775,A -85,B 0,C 180,E1 -20428.158,E2 -20428.158} C_VEL
LIN {X 0,Y 218.538,Z 400.004,A -85,B 0,C 180,E1 -20430.001,E2 -20430.001} C_VEL
LIN {X 0,Y 218.505,Z 399.81,A -85,B 0,C 180,E1 -20431.844,E2 -20431.844} C_VEL
LIN {X 0,Y 218.774,Z 398.246,A -85,B 0,C 180,E1 -20435.531,E2 -20435.531} C_VEL
LIN {X 0,Y 219.042,Z 396.882,A -85,B 0,C 180,E1 -20437.374,E2 -20437.374} C_VEL
LIN {X 0,Y 219.772,Z 393.998,A -85,B 0,C 180,E1 -20440.131,E2 -20440.131} C_VEL
LIN {X 0,Y 220.795,Z 390.09,A -85,B 0,C 180,E1 -20442.875,E2 -20442.875} C_VEL
LIN {X 0,Y 222.244,Z 385.05,A -85,B 0,C 180,E1 -20445.593,E2 -20445.593} C_VEL
LIN {X 0,Y 224.225,Z 378.703,A -85,B 0,C 180,E1 -20448.267,E2 -20448.267} C_VEL
LIN {X 0,Y 226.519,Z 370.765,A -85,B 0,C 180,E1 -20450.904,E2 -20450.904} C_VEL
LIN {X 0,Y 228.723,Z 362.566,A -85,B 0,C 180,E1 -20453.094,E2 -20453.094} C_VEL
LIN {X 0,Y 231.216,Z 352.802,A -85,B 0,C 180,E1 -20455.185,E2 -20455.185} C_VEL
LIN {X 0,Y 233.883,Z 341.688,A -85,B 0,C 180,E1 -20457.033,E2 -20457.033} C_VEL
LIN {X 0,Y 236.033,Z 330.795,A -85,B 0,C 180,E1 -20458.451,E2 -20458.451} C_VEL
LIN {X 0,Y 237.965,Z 318.756,A -85,B 0,C 180,E1 -20459.649,E2 -20459.649} C_VEL
LIN {X 0,Y 239.576,Z 305.766,A -85,B 0,C 180,E1 -20460.562,E2 -20460.562} C_VEL
LIN {X 0,Y 240.569,Z 293.038,A -85,B 0,C 180,E1 -20461.131,E2 -20461.131} C_VEL
LIN {X 0,Y 242.803,Z 234.276,A -85,B 0,C 180,E1 -20462.836,E2 -20462.836} C_VEL
LIN {X 0,Y 237.682,Z 220.938,A -85,B 0,C 180,E1 -20464.113,E2 -20464.113} C_VEL
LIN {X 0,Y 231.471,Z 207.573,A -85,B 0,C 180,E1 -20465.661,E2 -20465.661} C_VEL
LIN {X 0,Y 225.263,Z 195.648,A -85,B 0,C 180,E1 -20467.271,E2 -20467.271} C_VEL
LIN {X 0,Y 221.661,Z 188.981,A -85,B 0,C 180,E1 -20468.326,E2 -20468.326} C_VEL
LIN {X 0,Y 220.805,Z 186.014,A -85,B 0,C 180,E1 -20469.988,E2 -20469.988} C_VEL
LIN {X 0,Y 220.771,Z 185.965,A -85,B 0,C 180,E1 -20474.455,E2 -20474.455} C_VEL
LIN {X 0,Y 220.767,Z 185.951,A -85,B 0,C 180,E1 -20478.046,E2 -20478.046} C_VEL
LIN {X 0,Y 220.806,Z 185.982,A -85,B 0,C 180,E1 -20480.463,E2 -20480.463} C_VEL
LIN {X 0,Y 220.8,Z 185.923,A -85,B 0,C 180,E1 -20485.045,E2 -20485.045} C_VEL
LIN {X 0,Y 220.868,Z 185.973,A -85,B 0,C 180,E1 -20489.395,E2 -20489.395} C_VEL
LIN {X 0,Y 220.894,Z 185.959,A -85,B 0,C 180,E1 -20493.549,E2 -20493.549} C_VEL
LIN {X 0,Y 220.864,Z 185.955,A -85,B 0,C 180,E1 -20497.552,E2 -20497.552} C_VEL
LIN {X 0,Y 220.982,Z 185.949,A -85,B 0,C 180,E1 -20502.572,E2 -20502.572} C_VEL
LIN {X 0,Y 221.022,Z 185.951,A -85,B 0,C 180,E1 -20507.139,E2 -20507.139} C_VEL
LIN {X 0,Y 221.235,Z 185.901,A -85,B 0,C 180,E1 -20510.861,E2 -20510.861} C_VEL
LIN {X 0,Y 221.287,Z 185.909,A -85,B 0,C 180,E1 -20512.701,E2 -20512.701} C_VEL
LIN {X 0,Y 221.508,Z 185.87,A -85,B 0,C 180,E1 -20518.182,E2 -20518.182} C_VEL
LIN {X 0,Y 221.507,Z 185.891,A -85,B 0,C 180,E1 -20521.818,E2 -20521.818} C_VEL
LIN {X 0,Y 221.247,Z 185.922,A -85,B 0,C 180,E1 -20527.3,E2 -20527.3} C_VEL
LIN {X 0,Y 221.051,Z 185.928,A -85,B 0,C 180,E1 -20530.997,E2 -20530.997} C_VEL
LIN {X 0,Y 220.989,Z 185.943,A -85,B 0,C 180,E1 -20536.632,E2 -20536.632} C_VEL
LIN {X 0,Y 220.875,Z 185.971,A -85,B 0,C 180,E1 -20540.488,E2 -20540.488} C_VEL
LIN {X 0,Y 220.86,Z 185.957,A -85,B 0,C 180,E1 -20544.436,E2 -20544.436} C_VEL
LIN {X 0,Y 220.826,Z 185.966,A -85,B 0,C 180,E1 -20548.515,E2 -20548.515} C_VEL
LIN {X 0,Y 220.815,Z 185.976,A -85,B 0,C 180,E1 -20552.756,E2 -20552.756} C_VEL
LIN {X 0,Y 220.805,Z 185.951,A -85,B 0,C 180,E1 -20554.126,E2 -20554.126} C_VEL
LIN {X 0,Y 220.521,Z 185.978,A -85,B 0,C 180,E1 -20555.143,E2 -20555.143} C_VEL
LIN {X 0,Y 219.188,Z 186.145,A -85,B 0,C 180,E1 -20556.646,E2 -20556.646} C_VEL
LIN {X 0,Y 214.815,Z 186.722,A -85,B 0,C 180,E1 -20560.155,E2 -20560.155} C_VEL
LIN {X 0,Y 213.744,Z 186.853,A -85,B 0,C 180,E1 -20561.731,E2 -20561.731} C_VEL
LIN {X 0,Y 213.655,Z 186.859,A -85,B 0,C 180,E1 -20562.266,E2 -20562.266} C_VEL
LIN {X 0,Y 213.737,Z 186.942,A -85,B 0,C 180,E1 -20567.409,E2 -20567.409} C_VEL
LIN {X 0,Y 215.084,Z 191.907,A -85,B 0,C 180,E1 -20570.3,E2 -20570.3} C_VEL
LIN {X 0,Y 217.545,Z 196.431,A -85,B 0,C 180,E1 -20571.112,E2 -20571.112} C_VEL
LIN {X 0,Y 224.806,Z 210.156,A -85,B 0,C 180,E1 -20573.126,E2 -20573.126} C_VEL
LIN {X 0,Y 232.038,Z 226.341,A -85,B 0,C 180,E1 -20575.052,E2 -20575.052} C_VEL
LIN {X 0,Y 235.493,Z 235.427,A -85,B 0,C 180,E1 -20575.965,E2 -20575.965} C_VEL
LIN {X 0,Y 236.62,Z 243.856,A -85,B 0,C 180,E1 -20576.45,E2 -20576.45} C_VEL
LIN {X 0,Y 234.197,Z 300.703,A -85,B 0,C 180,E1 -20578.155,E2 -20578.155} C_VEL
LIN {X 0,Y 232.886,Z 313.646,A -85,B 0,C 180,E1 -20578.841,E2 -20578.841} C_VEL
LIN {X 0,Y 230.923,Z 326.557,A -85,B 0,C 180,E1 -20579.856,E2 -20579.856} C_VEL
LIN {X 0,Y 228.934,Z 337.634,A -85,B 0,C 180,E1 -20581.085,E2 -20581.085} C_VEL
LIN {X 0,Y 226.362,Z 349.179,A -85,B 0,C 180,E1 -20582.745,E2 -20582.745} C_VEL
LIN {X 0,Y 223.696,Z 359.575,A -85,B 0,C 180,E1 -20584.655,E2 -20584.655} C_VEL
LIN {X 0,Y 221.326,Z 368.073,A -85,B 0,C 180,E1 -20586.614,E2 -20586.614} C_VEL
LIN {X 0,Y 219.242,Z 375.677,A -85,B 0,C 180,E1 -20588.781,E2 -20588.781} C_VEL
LIN {X 0,Y 216.785,Z 383.566,A -85,B 0,C 180,E1 -20591.573,E2 -20591.573} C_VEL
LIN {X 0,Y 214.452,Z 390.625,A -85,B 0,C 180,E1 -20594.8,E2 -20594.8} C_VEL
LIN {X 0,Y 213.129,Z 395.319,A -85,B 0,C 180,E1 -20597.623,E2 -20597.623} C_VEL
LIN {X 0,Y 212.204,Z 398.904,A -85,B 0,C 180,E1 -20600.468,E2 -20600.468} C_VEL
LIN {X 0,Y 211.814,Z 400.752,A -85,B 0,C 180,E1 -20602.373,E2 -20602.373} C_VEL
LIN {X 0,Y 211.42,Z 402.944,A -85,B 0,C 180,E1 -20605.758,E2 -20605.758} C_VEL
LIN {X 0,Y 211.38,Z 403.728,A -85,B 0,C 180,E1 -20608.094,E2 -20608.094} C_VEL
LIN {X 0,Y 211.435,Z 403.938,A -85,B 0,C 180,E1 -20609.999,E2 -20609.999} C_VEL
LIN {X 0,Y 211.38,Z 403.716,A -85,B 0,C 180,E1 -20611.904,E2 -20611.904} C_VEL
LIN {X 0,Y 211.419,Z 402.925,A -85,B 0,C 180,E1 -20614.24,E2 -20614.24} C_VEL
LIN {X 0,Y 211.815,Z 400.713,A -85,B 0,C 180,E1 -20617.626,E2 -20617.626} C_VEL
LIN {X 0,Y 212.475,Z 397.782,A -85,B 0,C 180,E1 -20620.481,E2 -20620.481} C_VEL
LIN {X 0,Y 213.545,Z 393.815,A -85,B 0,C 180,E1 -20623.318,E2 -20623.318} C_VEL
LIN {X 0,Y 215.376,Z 387.715,A -85,B 0,C 180,E1 -20626.589,E2 -20626.589} C_VEL
LIN {X 0,Y 217.522,Z 381.052,A -85,B 0,C 180,E1 -20629.339,E2 -20629.339} C_VEL
LIN {X 0,Y 220.14,Z 372.24,A -85,B 0,C 180,E1 -20632.206,E2 -20632.206} C_VEL
LIN {X 0,Y 222.291,Z 364.298,A -85,B 0,C 180,E1 -20634.267,E2 -20634.267} C_VEL
LIN {X 0,Y 225.116,Z 353.814,A -85,B 0,C 180,E1 -20636.414,E2 -20636.414} C_VEL
LIN {X 0,Y 227.888,Z 342.008,A -85,B 0,C 180,E1 -20638.303,E2 -20638.303} C_VEL
LIN {X 0,Y 230.288,Z 330.108,A -85,B 0,C 180,E1 -20639.729,E2 -20639.729} C_VEL
LIN {X 0,Y 232.195,Z 317.715,A -85,B 0,C 180,E1 -20640.839,E2 -20640.839} C_VEL
LIN {X 0,Y 233.691,Z 305.298,A -85,B 0,C 180,E1 -20641.603,E2 -20641.603} C_VEL
LIN {X 0,Y 234.552,Z 292.073,A -85,B 0,C 180,E1 -20642.104,E2 -20642.104} C_VEL
LIN {X 0,Y 236.469,Z 242.514,A -85,B 0,C 180,E1 -20643.564,E2 -20643.564} C_VEL
LIN {X 0,Y 235.12,Z 234.355,A -85,B 0,C 180,E1 -20644.076,E2 -20644.076} C_VEL
LIN {X 0,Y 229.914,Z 221.44,A -85,B 0,C 180,E1 -20645.438,E2 -20645.438} C_VEL
LIN {X 0,Y 222.857,Z 206.368,A -85,B 0,C 180,E1 -20647.331,E2 -20647.331} C_VEL
LIN {X 0,Y 217.114,Z 195.788,A -85,B 0,C 180,E1 -20648.932,E2 -20648.932} C_VEL
LIN {X 0,Y 215.072,Z 191.863,A -85,B 0,C 180,E1 -20649.651,E2 -20649.651} C_VEL
LIN {X 0,Y 213.73,Z 186.915,A -85,B 0,C 180,E1 -20652.552,E2 -20652.552} C_VEL
LIN {X 0,Y 213.698,Z 186.853,A -85,B 0,C 180,E1 -20656.344,E2 -20656.344} C_VEL
LIN {X 0,Y 213.711,Z 186.866,A -85,B 0,C 180,E1 -20659.142,E2 -20659.142} C_VEL
LIN {X 0,Y 213.738,Z 186.806,A -85,B 0,C 180,E1 -20663.711,E2 -20663.711} C_VEL
LIN {X 0,Y 213.775,Z 186.852,A -85,B 0,C 180,E1 -20668.73,E2 -20668.73} C_VEL
LIN {X 0,Y 213.82,Z 186.849,A -85,B 0,C 180,E1 -20672.602,E2 -20672.602} C_VEL
LIN {X 0,Y 213.812,Z 186.836,A -85,B 0,C 180,E1 -20676.973,E2 -20676.973} C_VEL
LIN {X 0,Y 213.914,Z 186.819,A -85,B 0,C 180,E1 -20682.801,E2 -20682.801} C_VEL
LIN {X 0,Y 213.937,Z 186.827,A -85,B 0,C 180,E1 -20686.706,E2 -20686.706} C_VEL
LIN {X 0,Y 214.16,Z 186.8,A -85,B 0,C 180,E1 -20690.556,E2 -20690.556} C_VEL
LIN {X 0,Y 214.218,Z 186.8,A -85,B 0,C 180,E1 -20692.459,E2 -20692.459} C_VEL
LIN {X 0,Y 214.435,Z 186.772,A -85,B 0,C 180,E1 -20698.122,E2 -20698.122} C_VEL
LIN {X 0,Y 214.542,Z 186.755,A -85,B 0,C 180,E1 -20700,E2 -20700} C_VEL
LIN {X 0,Y 214.436,Z 186.75,A -85,B 0,C 180,E1 -20701.878,E2 -20701.878} C_VEL
LIN {X 0,Y 214.219,Z 186.786,A -85,B 0,C 180,E1 -20707.541,E2 -20707.541} C_VEL
LIN {X 0,Y 214.037,Z 186.815,A -85,B 0,C 180,E1 -20711.362,E2 -20711.362} C_VEL
LIN {X 0,Y 213.924,Z 186.816,A -85,B 0,C 180,E1 -20715.238,E2 -20715.238} C_VEL
LIN {X 0,Y 213.861,Z 186.845,A -85,B 0,C 180,E1 -20719.185,E2 -20719.185} C_VEL
LIN {X 0,Y 213.841,Z 186.834,A -85,B 0,C 180,E1 -20723.228,E2 -20723.228} C_VEL
LIN {X 0,Y 213.823,Z 186.834,A -85,B 0,C 180,E1 -20727.451,E2 -20727.451} C_VEL
LIN {X 0,Y 213.772,Z 186.846,A -85,B 0,C 180,E1 -20731.737,E2 -20731.737} C_VEL
LIN {X 0,Y 213.738,Z 186.807,A -85,B 0,C 180,E1 -20736.29,E2 -20736.29} C_VEL
LIN {X 0,Y 213.706,Z 186.844,A -85,B 0,C 180,E1 -20741.127,E2 -20741.127} C_VEL
LIN {X 0,Y 213.699,Z 186.824,A -85,B 0,C 180,E1 -20743.681,E2 -20743.681} C_VEL
LIN {X 0,Y 213.7,Z 186.858,A -85,B 0,C 180,E1 -20746.346,E2 -20746.346} C_VEL
LIN {X 0,Y 213.724,Z 186.996,A -85,B 0,C 180,E1 -20749.141,E2 -20749.141} C_VEL
LIN {X 0,Y 214.374,Z 189.148,A -85,B 0,C 180,E1 -20750.3,E2 -20750.3} C_VEL
LIN {X 0,Y 220.434,Z 199.925,A -85,B 0,C 180,E1 -20752.101,E2 -20752.101} C_VEL
LIN {X 0,Y 227.342,Z 213.44,A -85,B 0,C 180,E1 -20753.968,E2 -20753.968} C_VEL
LIN {X 0,Y 233.54,Z 227.372,A -85,B 0,C 180,E1 -20755.581,E2 -20755.581} C_VEL
LIN {X 0,Y 236.77,Z 235.975,A -85,B 0,C 180,E1 -20756.424,E2 -20756.424} C_VEL
LIN {X 0,Y 234.27,Z 296.602,A -85,B 0,C 180,E1 -20758.243,E2 -20758.243} C_VEL
LIN {X 0,Y 232.841,Z 310.335,A -85,B 0,C 180,E1 -20758.965,E2 -20758.965} C_VEL
LIN {X 0,Y 231.128,Z 323.106,A -85,B 0,C 180,E1 -20760.013,E2 -20760.013} C_VEL
LIN {X 0,Y 228.919,Z 334.921,A -85,B 0,C 180,E1 -20761.336,E2 -20761.336} C_VEL
LIN {X 0,Y 226.409,Z 346.274,A -85,B 0,C 180,E1 -20763.002,E2 -20763.002} C_VEL
LIN {X 0,Y 223.815,Z 356.507,A -85,B 0,C 180,E1 -20764.92,E2 -20764.92} C_VEL
LIN {X 0,Y 221.143,Z 366.569,A -85,B 0,C 180,E1 -20767.357,E2 -20767.357} C_VEL
LIN {X 0,Y 218.785,Z 374.618,A -85,B 0,C 180,E1 -20769.8,E2 -20769.8} C_VEL
LIN {X 0,Y 216.417,Z 381.808,A -85,B 0,C 180,E1 -20772.52,E2 -20772.52} C_VEL
LIN {X 0,Y 214.895,Z 386.655,A -85,B 0,C 180,E1 -20774.834,E2 -20774.834} C_VEL
LIN {X 0,Y 213.444,Z 391.366,A -85,B 0,C 180,E1 -20777.643,E2 -20777.643} C_VEL
LIN {X 0,Y 212.46,Z 394.971,A -85,B 0,C 180,E1 -20780.481,E2 -20780.481} C_VEL
LIN {X 0,Y 212,Z 396.833,A -85,B 0,C 180,E1 -20782.381,E2 -20782.381} C_VEL
LIN {X 0,Y 211.571,Z 398.792,A -85,B 0,C 180,E1 -20785.238,E2 -20785.238} C_VEL
LIN {X 0,Y 211.414,Z 399.84,A -85,B 0,C 180,E1 -20788.096,E2 -20788.096} C_VEL
LIN {X 0,Y 211.44,Z 400.069,A -85,B 0,C 180,E1 -20790.001,E2 -20790.001} C_VEL
LIN {X 0,Y 211.413,Z 399.874,A -85,B 0,C 180,E1 -20791.906,E2 -20791.906} C_VEL
LIN {X 0,Y 211.703,Z 398.311,A -85,B 0,C 180,E1 -20795.716,E2 -20795.716} C_VEL
LIN {X 0,Y 211.992,Z 396.946,A -85,B 0,C 180,E1 -20797.621,E2 -20797.621} C_VEL
LIN {X 0,Y 212.78,Z 394.062,A -85,B 0,C 180,E1 -20800.467,E2 -20800.467} C_VEL
LIN {X 0,Y 213.853,Z 390.154,A -85,B 0,C 180,E1 -20803.3,E2 -20803.3} C_VEL
LIN {X 0,Y 215.397,Z 385.114,A -85,B 0,C 180,E1 -20806.102,E2 -20806.102} C_VEL
LIN {X 0,Y 217.487,Z 378.766,A -85,B 0,C 180,E1 -20808.854,E2 -20808.854} C_VEL
LIN {X 0,Y 219.894,Z 370.827,A -85,B 0,C 180,E1 -20811.565,E2 -20811.565} C_VEL
LIN {X 0,Y 222.663,Z 360.955,A -85,B 0,C 180,E1 -20814.225,E2 -20814.225} C_VEL
LIN {X 0,Y 225.42,Z 350.589,A -85,B 0,C 180,E1 -20816.377,E2 -20816.377} C_VEL
LIN {X 0,Y 228.225,Z 338.899,A -85,B 0,C 180,E1 -20818.259,E2 -20818.259} C_VEL
LIN {X 0,Y 230.494,Z 327.238,A -85,B 0,C 180,E1 -20819.701,E2 -20819.701} C_VEL
LIN {X 0,Y 232.344,Z 315.108,A -85,B 0,C 180,E1 -20820.819,E2 -20820.819} C_VEL
LIN {X 0,Y 233.885,Z 301.872,A -85,B 0,C 180,E1 -20821.661,E2 -20821.661} C_VEL
LIN {X 0,Y 234.709,Z 288.295,A -85,B 0,C 180,E1 -20822.187,E2 -20822.187} C_VEL
LIN {X 0,Y 236.824,Z 235.852,A -85,B 0,C 180,E1 -20823.719,E2 -20823.719} C_VEL
LIN {X 0,Y 231.336,Z 222.045,A -85,B 0,C 180,E1 -20825.145,E2 -20825.145} C_VEL
LIN {X 0,Y 224.527,Z 207.663,A -85,B 0,C 180,E1 -20826.942,E2 -20826.942} C_VEL
LIN {X 0,Y 218.882,Z 197.094,A -85,B 0,C 180,E1 -20828.496,E2 -20828.496} C_VEL
LIN {X 0,Y 215.825,Z 191.965,A -85,B 0,C 180,E1 -20829.361,E2 -20829.361} C_VEL
LIN {X 0,Y 214.258,Z 188.789,A -85,B 0,C 180,E1 -20829.984,E2 -20829.984} C_VEL
LIN {X 0,Y 213.739,Z 186.914,A -85,B 0,C 180,E1 -20831.119,E2 -20831.119} C_VEL
LIN {X 0,Y 213.704,Z 186.861,A -85,B 0,C 180,E1 -20833.679,E2 -20833.679} C_VEL
LIN {X 0,Y 213.703,Z 186.824,A -85,B 0,C 180,E1 -20836.345,E2 -20836.345} C_VEL
LIN {X 0,Y 213.716,Z 186.845,A -85,B 0,C 180,E1 -20839.143,E2 -20839.143} C_VEL
LIN {X 0,Y 213.743,Z 186.807,A -85,B 0,C 180,E1 -20843.711,E2 -20843.711} C_VEL
LIN {X 0,Y 213.795,Z 186.847,A -85,B 0,C 180,E1 -20848.725,E2 -20848.725} C_VEL
LIN {X 0,Y 213.826,Z 186.833,A -85,B 0,C 180,E1 -20852.603,E2 -20852.603} C_VEL
LIN {X 0,Y 213.818,Z 186.836,A -85,B 0,C 180,E1 -20856.974,E2 -20856.974} C_VEL
LIN {X 0,Y 213.941,Z 186.822,A -85,B 0,C 180,E1 -20862.803,E2 -20862.803} C_VEL
LIN {X 0,Y 213.976,Z 186.828,A -85,B 0,C 180,E1 -20866.708,E2 -20866.708} C_VEL
LIN {X 0,Y 214.166,Z 186.782,A -85,B 0,C 180,E1 -20870.556,E2 -20870.556} C_VEL
LIN {X 0,Y 214.225,Z 186.785,A -85,B 0,C 180,E1 -20872.459,E2 -20872.459} C_VEL
LIN {X 0,Y 214.441,Z 186.749,A -85,B 0,C 180,E1 -20878.122,E2 -20878.122} C_VEL
LIN {X 0,Y 214.543,Z 186.754,A -85,B 0,C 180,E1 -20880,E2 -20880} C_VEL
LIN {X 0,Y 214.44,Z 186.771,A -85,B 0,C 180,E1 -20881.878,E2 -20881.878} C_VEL
LIN {X 0,Y 214.186,Z 186.804,A -85,B 0,C 180,E1 -20887.542,E2 -20887.542} C_VEL
LIN {X 0,Y 213.986,Z 186.807,A -85,B 0,C 180,E1 -20891.365,E2 -20891.365} C_VEL
LIN {X 0,Y 213.906,Z 186.839,A -85,B 0,C 180,E1 -20895.239,E2 -20895.239} C_VEL
LIN {X 0,Y 213.818,Z 186.837,A -85,B 0,C 180,E1 -20899.189,E2 -20899.189} C_VEL
LIN {X 0,Y 213.809,Z 186.835,A -85,B 0,C 180,E1 -20903.231,E2 -20903.231} C_VEL
LIN {X 0,Y 213.829,Z 186.847,A -85,B 0,C 180,E1 -20907.45,E2 -20907.45} C_VEL
LIN {X 0,Y 213.767,Z 186.859,A -85,B 0,C 180,E1 -20911.738,E2 -20911.738} C_VEL
LIN {X 0,Y 213.743,Z 186.806,A -85,B 0,C 180,E1 -20916.289,E2 -20916.289} C_VEL
LIN {X 0,Y 213.711,Z 186.864,A -85,B 0,C 180,E1 -20921.126,E2 -20921.126} C_VEL
LIN {X 0,Y 213.655,Z 186.859,A -85,B 0,C 180,E1 -20922.266,E2 -20922.266} C_VEL
LIN {X 0,Y 212.969,Z 186.943,A -85,B 0,C 180,E1 -20923.334,E2 -20923.334} C_VEL
LIN {X 0,Y 210.175,Z 187.451,A -85,B 0,C 180,E1 -20925.019,E2 -20925.019} C_VEL
LIN {X 0,Y 207.634,Z 188.825,A -85,B 0,C 180,E1 -20926.698,E2 -20926.698} C_VEL
LIN {X 0,Y 207.336,Z 190.221,A -85,B 0,C 180,E1 -20927.725,E2 -20927.725} C_VEL
LIN {X 0,Y 207.932,Z 192.153,A -85,B 0,C 180,E1 -20928.697,E2 -20928.697} C_VEL
LIN {X 0,Y 214.397,Z 203.64,A -85,B 0,C 180,E1 -20930.737,E2 -20930.737} C_VEL
LIN {X 0,Y 220.874,Z 216.345,A -85,B 0,C 180,E1 -20932.606,E2 -20932.606} C_VEL
LIN {X 0,Y 227.509,Z 231.623,A -85,B 0,C 180,E1 -20934.454,E2 -20934.454} C_VEL
LIN {X 0,Y 229.86,Z 238.126,A -85,B 0,C 180,E1 -20935.113,E2 -20935.113} C_VEL
LIN {X 0,Y 230.68,Z 245.125,A -85,B 0,C 180,E1 -20935.514,E2 -20935.514} C_VEL
LIN {X 0,Y 228.219,Z 300.435,A -85,B 0,C 180,E1 -20937.206,E2 -20937.206} C_VEL
LIN {X 0,Y 226.826,Z 313.725,A -85,B 0,C 180,E1 -20937.922,E2 -20937.922} C_VEL
LIN {X 0,Y 224.816,Z 326.498,A -85,B 0,C 180,E1 -20938.948,E2 -20938.948} C_VEL
LIN {X 0,Y 222.746,Z 337.574,A -85,B 0,C 180,E1 -20940.202,E2 -20940.202} C_VEL
LIN {X 0,Y 220.084,Z 349.118,A -85,B 0,C 180,E1 -20941.9,E2 -20941.9} C_VEL
LIN {X 0,Y 217.289,Z 359.513,A -85,B 0,C 180,E1 -20943.852,E2 -20943.852} C_VEL
LIN {X 0,Y 214.798,Z 368.01,A -85,B 0,C 180,E1 -20945.858,E2 -20945.858} C_VEL
LIN {X 0,Y 212.095,Z 377.22,A -85,B 0,C 180,E1 -20948.623,E2 -20948.623} C_VEL
LIN {X 0,Y 209.659,Z 384.62,A -85,B 0,C 180,E1 -20951.43,E2 -20951.43} C_VEL
LIN {X 0,Y 207.583,Z 390.561,A -85,B 0,C 180,E1 -20954.285,E2 -20954.285} C_VEL
LIN {X 0,Y 206.183,Z 395.255,A -85,B 0,C 180,E1 -20957.199,E2 -20957.199} C_VEL
LIN {X 0,Y 205.178,Z 398.839,A -85,B 0,C 180,E1 -20960.138,E2 -20960.138} C_VEL
LIN {X 0,Y 204.75,Z 400.687,A -85,B 0,C 180,E1 -20962.108,E2 -20962.108} C_VEL
LIN {X 0,Y 204.496,Z 402.072,A -85,B 0,C 180,E1 -20964.081,E2 -20964.081} C_VEL
LIN {X 0,Y 204.337,Z 403.061,A -85,B 0,C 180,E1 -20966.055,E2 -20966.055} C_VEL
LIN {X 0,Y 204.289,Z 403.663,A -85,B 0,C 180,E1 -20968.028,E2 -20968.028} C_VEL
LIN {X 0,Y 204.339,Z 403.873,A -85,B 0,C 180,E1 -20969.999,E2 -20969.999} C_VEL
LIN {X 0,Y 204.289,Z 403.651,A -85,B 0,C 180,E1 -20971.971,E2 -20971.971} C_VEL
LIN {X 0,Y 204.346,Z 402.96,A -85,B 0,C 180,E1 -20974.143,E2 -20974.143} C_VEL
LIN {X 0,Y 204.751,Z 400.648,A -85,B 0,C 180,E1 -20977.891,E2 -20977.891} C_VEL
LIN {X 0,Y 205.479,Z 397.716,A -85,B 0,C 180,E1 -20980.842,E2 -20980.842} C_VEL
LIN {X 0,Y 206.621,Z 393.749,A -85,B 0,C 180,E1 -20983.773,E2 -20983.773} C_VEL
LIN {X 0,Y 208.572,Z 387.648,A -85,B 0,C 180,E1 -20987.146,E2 -20987.146} C_VEL
LIN {X 0,Y 210.782,Z 380.985,A -85,B 0,C 180,E1 -20989.983,E2 -20989.983} C_VEL
LIN {X 0,Y 213.394,Z 372.745,A -85,B 0,C 180,E1 -20992.755,E2 -20992.755} C_VEL
LIN {X 0,Y 215.832,Z 364.23,A -85,B 0,C 180,E1 -20995.042,E2 -20995.042} C_VEL
LIN {X 0,Y 218.783,Z 353.746,A -85,B 0,C 180,E1 -20997.241,E2 -20997.241} C_VEL
LIN {X 0,Y 221.668,Z 341.939,A -85,B 0,C 180,E1 -20999.172,E2 -20999.172} C_VEL
LIN {X 0,Y 224.157,Z 330.037,A -85,B 0,C 180,E1 -21000.628,E2 -21000.628} C_VEL
LIN {X 0,Y 226.119,Z 317.642,A -85,B 0,C 180,E1 -21001.763,E2 -21001.763} C_VEL
LIN {X 0,Y 227.72,Z 304.896,A -85,B 0,C 180,E1 -21002.554,E2 -21002.554} C_VEL
LIN {X 0,Y 228.618,Z 290.516,A -85,B 0,C 180,E1 -21003.096,E2 -21003.096} C_VEL
LIN {X 0,Y 230.553,Z 243.441,A -85,B 0,C 180,E1 -21004.508,E2 -21004.508} C_VEL
LIN {X 0,Y 229.378,Z 236.69,A -85,B 0,C 180,E1 -21004.961,E2 -21004.961} C_VEL
LIN {X 0,Y 223.429,Z 222.138,A -85,B 0,C 180,E1 -21006.6,E2 -21006.6} C_VEL
LIN {X 0,Y 216.993,Z 208.549,A -85,B 0,C 180,E1 -21008.428,E2 -21008.428} C_VEL
LIN {X 0,Y 210.249,Z 196.263,A -85,B 0,C 180,E1 -21010.434,E2 -21010.434} C_VEL
LIN {X 0,Y 207.828,Z 191.917,A -85,B 0,C 180,E1 -21011.282,E2 -21011.282} C_VEL
LIN {X 0,Y 206.662,Z 187.845,A -85,B 0,C 180,E1 -21013.757,E2 -21013.757} C_VEL
LIN {X 0,Y 206.636,Z 187.741,A -85,B 0,C 180,E1 -21018.436,E2 -21018.436} C_VEL
LIN {X 0,Y 206.673,Z 187.689,A -85,B 0,C 180,E1 -21022.259,E2 -21022.259} C_VEL
LIN {X 0,Y 206.693,Z 187.733,A -85,B 0,C 180,E1 -21027.041,E2 -21027.041} C_VEL
LIN {X 0,Y 206.758,Z 187.724,A -85,B 0,C 180,E1 -21032.097,E2 -21032.097} C_VEL
LIN {X 0,Y 206.747,Z 187.713,A -85,B 0,C 180,E1 -21036.604,E2 -21036.604} C_VEL
LIN {X 0,Y 206.861,Z 187.696,A -85,B 0,C 180,E1 -21042.196,E2 -21042.196} C_VEL
LIN {X 0,Y 206.878,Z 187.71,A -85,B 0,C 180,E1 -21046.243,E2 -21046.243} C_VEL
LIN {X 0,Y 207.098,Z 187.675,A -85,B 0,C 180,E1 -21050.231,E2 -21050.231} C_VEL
LIN {X 0,Y 207.159,Z 187.681,A -85,B 0,C 180,E1 -21052.201,E2 -21052.201} C_VEL
LIN {X 0,Y 207.372,Z 187.651,A -85,B 0,C 180,E1 -21058.058,E2 -21058.058} C_VEL
LIN {X 0,Y 207.507,Z 187.631,A -85,B 0,C 180,E1 -21060,E2 -21060} C_VEL
LIN {X 0,Y 207.372,Z 187.629,A -85,B 0,C 180,E1 -21061.942,E2 -21061.942} C_VEL
LIN {X 0,Y 207.16,Z 187.662,A -85,B 0,C 180,E1 -21067.799,E2 -21067.799} C_VEL
LIN {X 0,Y 206.974,Z 187.699,A -85,B 0,C 180,E1 -21071.756,E2 -21071.756} C_VEL
LIN {X 0,Y 206.858,Z 187.694,A -85,B 0,C 180,E1 -21075.772,E2 -21075.772} C_VEL
LIN {X 0,Y 206.793,Z 187.722,A -85,B 0,C 180,E1 -21079.868,E2 -21079.868} C_VEL
LIN {X 0,Y 206.758,Z 187.726,A -85,B 0,C 180,E1 -21084.073,E2 -21084.073} C_VEL
LIN {X 0,Y 206.739,Z 187.717,A -85,B 0,C 180,E1 -21088.42,E2 -21088.42} C_VEL
LIN {X 0,Y 206.697,Z 187.698,A -85,B 0,C 180,E1 -21092.958,E2 -21092.958} C_VEL
LIN {X 0,Y 206.674,Z 187.706,A -85,B 0,C 180,E1 -21097.741,E2 -21097.741} C_VEL
LIN {X 0,Y 206.636,Z 187.716,A -85,B 0,C 180,E1 -21101.564,E2 -21101.564} C_VEL
LIN {X 0,Y 206.627,Z 187.722,A -85,B 0,C 180,E1 -21105.584,E2 -21105.584} C_VEL
LIN {X 0,Y 206.638,Z 187.907,A -85,B 0,C 180,E1 -21107.884,E2 -21107.884} C_VEL
LIN {X 0,Y 207.06,Z 189.374,A -85,B 0,C 180,E1 -21108.621,E2 -21108.621} C_VEL
LIN {X 0,Y 212.8,Z 198.961,A -85,B 0,C 180,E1 -21110.437,E2 -21110.437} C_VEL
LIN {X 0,Y 220.01,Z 212.505,A -85,B 0,C 180,E1 -21112.524,E2 -21112.524} C_VEL
LIN {X 0,Y 227.016,Z 227.891,A -85,B 0,C 180,E1 -21114.461,E2 -21114.461} C_VEL
LIN {X 0,Y 230.831,Z 237.734,A -85,B 0,C 180,E1 -21115.502,E2 -21115.502} C_VEL
LIN {X 0,Y 228.307,Z 296.463,A -85,B 0,C 180,E1 -21117.299,E2 -21117.299} C_VEL
LIN {X 0,Y 226.852,Z 309.844,A -85,B 0,C 180,E1 -21118.002,E2 -21118.002} C_VEL
LIN {X 0,Y 225.201,Z 322.092,A -85,B 0,C 180,E1 -21119.009,E2 -21119.009} C_VEL
LIN {X 0,Y 223.049,Z 333.407,A -85,B 0,C 180,E1 -21120.249,E2 -21120.249} C_VEL
LIN {X 0,Y 220.444,Z 345.053,A -85,B 0,C 180,E1 -21121.951,E2 -21121.951} C_VEL
LIN {X 0,Y 217.707,Z 355.517,A -85,B 0,C 180,E1 -21123.908,E2 -21123.908} C_VEL
LIN {X 0,Y 214.913,Z 365.479,A -85,B 0,C 180,E1 -21126.298,E2 -21126.298} C_VEL
LIN {X 0,Y 212.126,Z 374.686,A -85,B 0,C 180,E1 -21129.137,E2 -21129.137} C_VEL
LIN {X 0,Y 209.658,Z 381.875,A -85,B 0,C 180,E1 -21131.938,E2 -21131.938} C_VEL
LIN {X 0,Y 208.019,Z 386.721,A -85,B 0,C 180,E1 -21134.32,E2 -21134.32} C_VEL
LIN {X 0,Y 206.494,Z 391.432,A -85,B 0,C 180,E1 -21137.22,E2 -21137.22} C_VEL
LIN {X 0,Y 205.46,Z 395.036,A -85,B 0,C 180,E1 -21140.153,E2 -21140.153} C_VEL
LIN {X 0,Y 204.943,Z 396.898,A -85,B 0,C 180,E1 -21142.117,E2 -21142.117} C_VEL
LIN {X 0,Y 204.467,Z 399.034,A -85,B 0,C 180,E1 -21145.417,E2 -21145.417} C_VEL
LIN {X 0,Y 204.324,Z 399.905,A -85,B 0,C 180,E1 -21148.03,E2 -21148.03} C_VEL
LIN {X 0,Y 204.345,Z 400.134,A -85,B 0,C 180,E1 -21150.001,E2 -21150.001} C_VEL
LIN {X 0,Y 204.323,Z 399.939,A -85,B 0,C 180,E1 -21151.972,E2 -21151.972} C_VEL
LIN {X 0,Y 204.503,Z 399.04,A -85,B 0,C 180,E1 -21154.706,E2 -21154.706} C_VEL
LIN {X 0,Y 204.938,Z 397.01,A -85,B 0,C 180,E1 -21157.885,E2 -21157.885} C_VEL
LIN {X 0,Y 205.777,Z 394.127,A -85,B 0,C 180,E1 -21160.828,E2 -21160.828} C_VEL
LIN {X 0,Y 206.934,Z 390.218,A -85,B 0,C 180,E1 -21163.754,E2 -21163.754} C_VEL
LIN {X 0,Y 208.576,Z 385.177,A -85,B 0,C 180,E1 -21166.643,E2 -21166.643} C_VEL
LIN {X 0,Y 210.778,Z 378.829,A -85,B 0,C 180,E1 -21169.478,E2 -21169.478} C_VEL
LIN {X 0,Y 213.28,Z 370.963,A -85,B 0,C 180,E1 -21172.244,E2 -21172.244} C_VEL
LIN {X 0,Y 215.672,Z 362.8,A -85,B 0,C 180,E1 -21174.549,E2 -21174.549} C_VEL
LIN {X 0,Y 218.466,Z 352.925,A -85,B 0,C 180,E1 -21176.768,E2 -21176.768} C_VEL
LIN {X 0,Y 221.351,Z 341.808,A -85,B 0,C 180,E1 -21178.7,E2 -21178.7} C_VEL
LIN {X 0,Y 223.659,Z 330.913,A -85,B 0,C 180,E1 -21180.183,E2 -21180.183} C_VEL
LIN {X 0,Y 225.756,Z 318.871,A -85,B 0,C 180,E1 -21181.429,E2 -21181.429} C_VEL
LIN {X 0,Y 227.41,Z 306.543,A -85,B 0,C 180,E1 -21182.341,E2 -21182.341} C_VEL
LIN {X 0,Y 228.569,Z 292.757,A -85,B 0,C 180,E1 -21182.982,E2 -21182.982} C_VEL
LIN {X 0,Y 230.881,Z 237.764,A -85,B 0,C 180,E1 -21184.64,E2 -21184.64} C_VEL
LIN {X 0,Y 225.519,Z 224.225,A -85,B 0,C 180,E1 -21186.11,E2 -21186.11} C_VEL
LIN {X 0,Y 218.312,Z 209.106,A -85,B 0,C 180,E1 -21188.121,E2 -21188.121} C_VEL
LIN {X 0,Y 212.158,Z 197.811,A -85,B 0,C 180,E1 -21189.926,E2 -21189.926} C_VEL
LIN {X 0,Y 208.707,Z 192.265,A -85,B 0,C 180,E1 -21190.972,E2 -21190.972} C_VEL
LIN {X 0,Y 206.974,Z 188.977,A -85,B 0,C 180,E1 -21191.666,E2 -21191.666} C_VEL
LIN {X 0,Y 206.679,Z 187.777,A -85,B 0,C 180,E1 -21192.495,E2 -21192.495} C_VEL
LIN {X 0,Y 206.623,Z 187.705,A -85,B 0,C 180,E1 -21197.135,E2 -21197.135} C_VEL
LIN {X 0,Y 206.688,Z 187.727,A -85,B 0,C 180,E1 -21201.45,E2 -21201.45} C_VEL
LIN {X 0,Y 206.699,Z 187.678,A -85,B 0,C 180,E1 -21204.688,E2 -21204.688} C_VEL
LIN {X 0,Y 206.724,Z 187.734,A -85,B 0,C 180,E1 -21209.339,E2 -21209.339} C_VEL
LIN {X 0,Y 206.731,Z 187.724,A -85,B 0,C 180,E1 -21213.772,E2 -21213.772} C_VEL
LIN {X 0,Y 206.737,Z 187.713,A -85,B 0,C 180,E1 -21218.041,E2 -21218.041} C_VEL
LIN {X 0,Y 206.871,Z 187.71,A -85,B 0,C 180,E1 -21222.196,E2 -21222.196} C_VEL
LIN {X 0,Y 206.909,Z 187.701,A -85,B 0,C 180,E1 -21226.245,E2 -21226.245} C_VEL
LIN {X 0,Y 207.104,Z 187.662,A -85,B 0,C 180,E1 -21230.231,E2 -21230.231} C_VEL
LIN {X 0,Y 207.166,Z 187.66,A -85,B 0,C 180,E1 -21232.201,E2 -21232.201} C_VEL
LIN {X 0,Y 207.378,Z 187.628,A -85,B 0,C 180,E1 -21238.058,E2 -21238.058} C_VEL
LIN {X 0,Y 207.509,Z 187.63,A -85,B 0,C 180,E1 -21240,E2 -21240} C_VEL
LIN {X 0,Y 207.376,Z 187.651,A -85,B 0,C 180,E1 -21241.942,E2 -21241.942} C_VEL
LIN {X 0,Y 207.128,Z 187.685,A -85,B 0,C 180,E1 -21247.8,E2 -21247.8} C_VEL
LIN {X 0,Y 206.909,Z 187.688,A -85,B 0,C 180,E1 -21251.759,E2 -21251.759} C_VEL
LIN {X 0,Y 206.841,Z 187.715,A -85,B 0,C 180,E1 -21255.773,E2 -21255.773} C_VEL
LIN {X 0,Y 206.856,Z 187.696,A -85,B 0,C 180,E1 -21257.955,E2 -21257.955} C_VEL
LIN {X 0,Y 206.752,Z 187.713,A -85,B 0,C 180,E1 -21263.395,E2 -21263.395} C_VEL
LIN {X 0,Y 206.736,Z 187.721,A -85,B 0,C 180,E1 -21268.42,E2 -21268.42} C_VEL
LIN {X 0,Y 206.698,Z 187.731,A -85,B 0,C 180,E1 -21272.958,E2 -21272.958} C_VEL
LIN {X 0,Y 206.678,Z 187.69,A -85,B 0,C 180,E1 -21277.74,E2 -21277.74} C_VEL
LIN {X 0,Y 206.617,Z 187.735,A -85,B 0,C 180,E1 -21282.26,E2 -21282.26} C_VEL
LIN {X 0,Y 206.695,Z 187.927,A -85,B 0,C 180,E1 -21286.243,E2 -21286.243} C_VEL
LIN {X 0,Y 207.336,Z 190.221,A -85,B 0,C 180,E1 -21287.725,E2 -21287.725} C_VEL
LIN {X 0,Y 208.072,Z 192.35,A -85,B 0,C 180,E1 -21288.56,E2 -21288.56} C_VEL
LIN {X 0,Y 209.47,Z 196.068,A -85,B 0,C 180,E1 -21289.294,E2 -21289.294} C_VEL
LIN {X 0,Y 211.312,Z 202.242,A -85,B 0,C 180,E1 -21289.991,E2 -21289.991} C_VEL
LIN {X 0,Y 214.188,Z 215.989,A -85,B 0,C 180,E1 -21291.211,E2 -21291.211} C_VEL
LIN {X 0,Y 214.813,Z 217.83,A -85,B 0,C 180,E1 -21291.424,E2 -21291.424} C_VEL
LIN {X 0,Y 221.763,Z 233.86,A -85,B 0,C 180,E1 -21293.476,E2 -21293.476} C_VEL
LIN {X 0,Y 224.276,Z 240.845,A -85,B 0,C 180,E1 -21294.219,E2 -21294.219} C_VEL
LIN {X 0,Y 224.832,Z 246.316,A -85,B 0,C 180,E1 -21294.532,E2 -21294.532} C_VEL
LIN {X 0,Y 222.316,Z 300.24,A -85,B 0,C 180,E1 -21296.211,E2 -21296.211} C_VEL
LIN {X 0,Y 220.92,Z 313.146,A -85,B 0,C 180,E1 -21296.91,E2 -21296.91} C_VEL
LIN {X 0,Y 218.976,Z 325.335,A -85,B 0,C 180,E1 -21297.888,E2 -21297.888} C_VEL
LIN {X 0,Y 216.612,Z 337.513,A -85,B 0,C 180,E1 -21299.269,E2 -21299.269} C_VEL
LIN {X 0,Y 213.85,Z 349.057,A -85,B 0,C 180,E1 -21301.004,E2 -21301.004} C_VEL
LIN {X 0,Y 210.938,Z 359.451,A -85,B 0,C 180,E1 -21303.002,E2 -21303.002} C_VEL
LIN {X 0,Y 208.327,Z 367.948,A -85,B 0,C 180,E1 -21305.058,E2 -21305.058} C_VEL
LIN {X 0,Y 205.868,Z 376.084,A -85,B 0,C 180,E1 -21307.526,E2 -21307.526} C_VEL
LIN {X 0,Y 203.328,Z 383.439,A -85,B 0,C 180,E1 -21310.305,E2 -21310.305} C_VEL
LIN {X 0,Y 200.741,Z 390.497,A -85,B 0,C 180,E1 -21313.734,E2 -21313.734} C_VEL
LIN {X 0,Y 199.235,Z 395.191,A -85,B 0,C 180,E1 -21316.744,E2 -21316.744} C_VEL
LIN {X 0,Y 198.174,Z 398.775,A -85,B 0,C 180,E1 -21319.786,E2 -21319.786} C_VEL
LIN {X 0,Y 197.703,Z 400.622,A -85,B 0,C 180,E1 -21321.825,E2 -21321.825} C_VEL
LIN {X 0,Y 197.411,Z 402.007,A -85,B 0,C 180,E1 -21323.868,E2 -21323.868} C_VEL
LIN {X 0,Y 197.24,Z 403.072,A -85,B 0,C 180,E1 -21326.106,E2 -21326.106} C_VEL
LIN {X 0,Y 197.246,Z 403.808,A -85,B 0,C 180,E1 -21329.999,E2 -21329.999} C_VEL
LIN {X 0,Y 197.235,Z 403.059,A -85,B 0,C 180,E1 -21333.874,E2 -21333.874} C_VEL
LIN {X 0,Y 197.411,Z 401.979,A -85,B 0,C 180,E1 -21336.13,E2 -21336.13} C_VEL
LIN {X 0,Y 197.704,Z 400.582,A -85,B 0,C 180,E1 -21338.174,E2 -21338.174} C_VEL
LIN {X 0,Y 198.486,Z 397.65,A -85,B 0,C 180,E1 -21341.229,E2 -21341.229} C_VEL
LIN {X 0,Y 199.687,Z 393.683,A -85,B 0,C 180,E1 -21344.261,E2 -21344.261} C_VEL
LIN {X 0,Y 201.775,Z 387.581,A -85,B 0,C 180,E1 -21347.743,E2 -21347.743} C_VEL
LIN {X 0,Y 204.083,Z 380.917,A -85,B 0,C 180,E1 -21350.668,E2 -21350.668} C_VEL
LIN {X 0,Y 206.611,Z 373.359,A -85,B 0,C 180,E1 -21353.303,E2 -21353.303} C_VEL
LIN {X 0,Y 209.407,Z 364.162,A -85,B 0,C 180,E1 -21355.866,E2 -21355.866} C_VEL
LIN {X 0,Y 212.492,Z 353.677,A -85,B 0,C 180,E1 -21358.118,E2 -21358.118} C_VEL
LIN {X 0,Y 215.136,Z 343.298,A -85,B 0,C 180,E1 -21359.878,E2 -21359.878} C_VEL
LIN {X 0,Y 217.688,Z 331.908,A -85,B 0,C 180,E1 -21361.37,E2 -21361.37} C_VEL
LIN {X 0,Y 219.72,Z 320.171,A -85,B 0,C 180,E1 -21362.53,E2 -21362.53} C_VEL
LIN {X 0,Y 221.545,Z 306.903,A -85,B 0,C 180,E1 -21363.426,E2 -21363.426} C_VEL
LIN {X 0,Y 222.557,Z 293.756,A -85,B 0,C 180,E1 -21363.992,E2 -21363.992} C_VEL
LIN {X 0,Y 224.703,Z 244.54,A -85,B 0,C 180,E1 -21365.494,E2 -21365.494} C_VEL
LIN {X 0,Y 223.819,Z 239.441,A -85,B 0,C 180,E1 -21365.853,E2 -21365.853} C_VEL
LIN {X 0,Y 218.293,Z 225.747,A -85,B 0,C 180,E1 -21367.458,E2 -21367.458} C_VEL
LIN {X 0,Y 212.106,Z 212.483,A -85,B 0,C 180,E1 -21369.311,E2 -21369.311} C_VEL
LIN {X 0,Y 205.544,Z 200.489,A -85,B 0,C 180,E1 -21371.364,E2 -21371.364} C_VEL
LIN {X 0,Y 202.314,Z 195.236,A -85,B 0,C 180,E1 -21372.419,E2 -21372.419} C_VEL
LIN {X 0,Y 200.487,Z 191.747,A -85,B 0,C 180,E1 -21373.175,E2 -21373.175} C_VEL
LIN {X 0,Y 199.584,Z 188.654,A -85,B 0,C 180,E1 -21375.23,E2 -21375.23} C_VEL
LIN {X 0,Y 199.573,Z 188.615,A -85,B 0,C 180,E1 -21378.003,E2 -21378.003} C_VEL
LIN {X 0,Y 199.604,Z 188.589,A -85,B 0,C 180,E1 -21380.767,E2 -21380.767} C_VEL
LIN {X 0,Y 199.606,Z 188.585,A -85,B 0,C 180,E1 -21385.712,E2 -21385.712} C_VEL
LIN {X 0,Y 199.687,Z 188.612,A -85,B 0,C 180,E1 -21388.135,E2 -21388.135} C_VEL
LIN {X 0,Y 199.68,Z 188.612,A -85,B 0,C 180,E1 -21392.771,E2 -21392.771} C_VEL
LIN {X 0,Y 199.706,Z 188.594,A -85,B 0,C 180,E1 -21397.225,E2 -21397.225} C_VEL
LIN {X 0,Y 199.788,Z 188.576,A -85,B 0,C 180,E1 -21401.759,E2 -21401.759} C_VEL
LIN {X 0,Y 199.816,Z 188.595,A -85,B 0,C 180,E1 -21405.747,E2 -21405.747} C_VEL
LIN {X 0,Y 200.064,Z 188.547,A -85,B 0,C 180,E1 -21409.884,E2 -21409.884} C_VEL
LIN {X 0,Y 200.023,Z 188.551,A -85,B 0,C 180,E1 -21413.949,E2 -21413.949} C_VEL
LIN {X 0,Y 200.311,Z 188.531,A -85,B 0,C 180,E1 -21417.989,E2 -21417.989} C_VEL
LIN {X 0,Y 200.471,Z 188.507,A -85,B 0,C 180,E1 -21420,E2 -21420} C_VEL
LIN {X 0,Y 200.019,Z 188.554,A -85,B 0,C 180,E1 -21424.03,E2 -21424.03} C_VEL
LIN {X 0,Y 200.104,Z 188.537,A -85,B 0,C 180,E1 -21428.076,E2 -21428.076} C_VEL
LIN {X 0,Y 199.906,Z 188.581,A -85,B 0,C 180,E1 -21432.178,E2 -21432.178} C_VEL
LIN {X 0,Y 199.797,Z 188.575,A -85,B 0,C 180,E1 -21436.344,E2 -21436.344} C_VEL
LIN {X 0,Y 199.818,Z 188.593,A -85,B 0,C 180,E1 -21438.454,E2 -21438.454} C_VEL
LIN {X 0,Y 199.731,Z 188.597,A -85,B 0,C 180,E1 -21443.818,E2 -21443.818} C_VEL
LIN {X 0,Y 199.707,Z 188.592,A -85,B 0,C 180,E1 -21448.388,E2 -21448.388} C_VEL
LIN {X 0,Y 199.672,Z 188.583,A -85,B 0,C 180,E1 -21452.359,E2 -21452.359} C_VEL
LIN {X 0,Y 199.618,Z 188.568,A -85,B 0,C 180,E1 -21456.765,E2 -21456.765} C_VEL
LIN {X 0,Y 199.604,Z 188.621,A -85,B 0,C 180,E1 -21459.329,E2 -21459.329} C_VEL
LIN {X 0,Y 199.568,Z 188.587,A -85,B 0,C 180,E1 -21462.311,E2 -21462.311} C_VEL
LIN {X 0,Y 199.589,Z 188.822,A -85,B 0,C 180,E1 -21466.358,E2 -21466.358} C_VEL
LIN {X 0,Y 199.81,Z 189.759,A -85,B 0,C 180,E1 -21466.784,E2 -21466.784} C_VEL
LIN {X 0,Y 201.552,Z 192.748,A -85,B 0,C 180,E1 -21467.439,E2 -21467.439} C_VEL
LIN {X 0,Y 203.429,Z 195.469,A -85,B 0,C 180,E1 -21468.051,E2 -21468.051} C_VEL
LIN {X 0,Y 208.807,Z 204.504,A -85,B 0,C 180,E1 -21469.768,E2 -21469.768} C_VEL
LIN {X 0,Y 215.193,Z 216.693,A -85,B 0,C 180,E1 -21471.706,E2 -21471.706} C_VEL
LIN {X 0,Y 222.357,Z 232.739,A -85,B 0,C 180,E1 -21473.787,E2 -21473.787} C_VEL
LIN {X 0,Y 224.964,Z 239.642,A -85,B 0,C 180,E1 -21474.539,E2 -21474.539} C_VEL
LIN {X 0,Y 222.381,Z 296.445,A -85,B 0,C 180,E1 -21476.307,E2 -21476.307} C_VEL
LIN {X 0,Y 220.862,Z 310.024,A -85,B 0,C 180,E1 -21477.035,E2 -21477.035} C_VEL
LIN {X 0,Y 219.157,Z 322.164,A -85,B 0,C 180,E1 -21478.055,E2 -21478.055} C_VEL
LIN {X 0,Y 216.915,Z 333.477,A -85,B 0,C 180,E1 -21479.318,E2 -21479.318} C_VEL
LIN {X 0,Y 214.222,Z 345.122,A -85,B 0,C 180,E1 -21481.061,E2 -21481.061} C_VEL
LIN {X 0,Y 211.335,Z 355.585,A -85,B 0,C 180,E1 -21483.059,E2 -21483.059} C_VEL
LIN {X 0,Y 208.543,Z 365.179,A -85,B 0,C 180,E1 -21485.408,E2 -21485.408} C_VEL
LIN {X 0,Y 205.909,Z 373.402,A -85,B 0,C 180,E1 -21487.95,E2 -21487.95} C_VEL
LIN {X 0,Y 203.332,Z 380.828,A -85,B 0,C 180,E1 -21490.832,E2 -21490.832} C_VEL
LIN {X 0,Y 201.165,Z 386.788,A -85,B 0,C 180,E1 -21493.771,E2 -21493.771} C_VEL
LIN {X 0,Y 199.565,Z 391.498,A -85,B 0,C 180,E1 -21496.768,E2 -21496.768} C_VEL
LIN {X 0,Y 198.448,Z 395.102,A -85,B 0,C 180,E1 -21499.802,E2 -21499.802} C_VEL
LIN {X 0,Y 197.913,Z 396.964,A -85,B 0,C 180,E1 -21501.835,E2 -21501.835} C_VEL
LIN {X 0,Y 197.371,Z 399.228,A -85,B 0,C 180,E1 -21505.584,E2 -21505.584} C_VEL
LIN {X 0,Y 197.236,Z 399.97,A -85,B 0,C 180,E1 -21507.959,E2 -21507.959} C_VEL
LIN {X 0,Y 197.252,Z 400.199,A -85,B 0,C 180,E1 -21510.001,E2 -21510.001} C_VEL
LIN {X 0,Y 197.236,Z 400.004,A -85,B 0,C 180,E1 -21512.043,E2 -21512.043} C_VEL
LIN {X 0,Y 197.406,Z 399.234,A -85,B 0,C 180,E1 -21514.544,E2 -21514.544} C_VEL
LIN {X 0,Y 197.91,Z 397.075,A -85,B 0,C 180,E1 -21518.167,E2 -21518.167} C_VEL
LIN {X 0,Y 198.796,Z 394.191,A -85,B 0,C 180,E1 -21521.213,E2 -21521.213} C_VEL
LIN {X 0,Y 200.037,Z 390.282,A -85,B 0,C 180,E1 -21524.238,E2 -21524.238} C_VEL
LIN {X 0,Y 201.782,Z 385.241,A -85,B 0,C 180,E1 -21527.221,E2 -21527.221} C_VEL
LIN {X 0,Y 204.1,Z 378.892,A -85,B 0,C 180,E1 -21530.142,E2 -21530.142} C_VEL
LIN {X 0,Y 206.98,Z 370.277,A -85,B 0,C 180,E1 -21533.226,E2 -21533.226} C_VEL
LIN {X 0,Y 209.751,Z 361.08,A -85,B 0,C 180,E1 -21535.823,E2 -21535.823} C_VEL
LIN {X 0,Y 212.809,Z 350.711,A -85,B 0,C 180,E1 -21538.074,E2 -21538.074} C_VEL
LIN {X 0,Y 215.819,Z 339.019,A -85,B 0,C 180,E1 -21540.045,E2 -21540.045} C_VEL
LIN {X 0,Y 218.308,Z 327.355,A -85,B 0,C 180,E1 -21541.543,E2 -21541.543} C_VEL
LIN {X 0,Y 220.28,Z 315.22,A -85,B 0,C 180,E1 -21542.71,E2 -21542.71} C_VEL
LIN {X 0,Y 221.913,Z 302.193,A -85,B 0,C 180,E1 -21543.572,E2 -21543.572} C_VEL
LIN {X 0,Y 222.791,Z 290.156,A -85,B 0,C 180,E1 -21544.07,E2 -21544.07} C_VEL
LIN {X 0,Y 225,Z 239.677,A -85,B 0,C 180,E1 -21545.609,E2 -21545.609} C_VEL
LIN {X 0,Y 219.725,Z 226.343,A -85,B 0,C 180,E1 -21547.136,E2 -21547.136} C_VEL
LIN {X 0,Y 212.231,Z 210.679,A -85,B 0,C 180,E1 -21549.355,E2 -21549.355} C_VEL
LIN {X 0,Y 206.676,Z 200.837,A -85,B 0,C 180,E1 -21551.075,E2 -21551.075} C_VEL
LIN {X 0,Y 201.997,Z 193.097,A -85,B 0,C 180,E1 -21552.61,E2 -21552.61} C_VEL
LIN {X 0,Y 200.251,Z 190.834,A -85,B 0,C 180,E1 -21553.185,E2 -21553.185} C_VEL
LIN {X 0,Y 199.686,Z 189.167,A -85,B 0,C 180,E1 -21553.589,E2 -21553.589} C_VEL
LIN {X 0,Y 199.609,Z 188.634,A -85,B 0,C 180,E1 -21554.3,E2 -21554.3} C_VEL
LIN {X 0,Y 199.578,Z 188.587,A -85,B 0,C 180,E1 -21558.004,E2 -21558.004} C_VEL
LIN {X 0,Y 199.612,Z 188.622,A -85,B 0,C 180,E1 -21560.767,E2 -21560.767} C_VEL
LIN {X 0,Y 199.613,Z 188.562,A -85,B 0,C 180,E1 -21565.713,E2 -21565.713} C_VEL
LIN {X 0,Y 199.7,Z 188.587,A -85,B 0,C 180,E1 -21568.137,E2 -21568.137} C_VEL
LIN {X 0,Y 199.686,Z 188.594,A -85,B 0,C 180,E1 -21572.771,E2 -21572.771} C_VEL
LIN {X 0,Y 199.713,Z 188.59,A -85,B 0,C 180,E1 -21577.226,E2 -21577.226} C_VEL
LIN {X 0,Y 199.795,Z 188.595,A -85,B 0,C 180,E1 -21581.758,E2 -21581.758} C_VEL
LIN {X 0,Y 199.844,Z 188.575,A -85,B 0,C 180,E1 -21585.749,E2 -21585.749} C_VEL
LIN {X 0,Y 200.07,Z 188.54,A -85,B 0,C 180,E1 -21589.884,E2 -21589.884} C_VEL
LIN {X 0,Y 200.03,Z 188.568,A -85,B 0,C 180,E1 -21593.949,E2 -21593.949} C_VEL
LIN {X 0,Y 200.317,Z 188.507,A -85,B 0,C 180,E1 -21597.989,E2 -21597.989} C_VEL
LIN {X 0,Y 200.474,Z 188.506,A -85,B 0,C 180,E1 -21600,E2 -21600} C_VEL
LIN {X 0,Y 200.017,Z 188.545,A -85,B 0,C 180,E1 -21604.03,E2 -21604.03} C_VEL
LIN {X 0,Y 200.074,Z 188.563,A -85,B 0,C 180,E1 -21608.077,E2 -21608.077} C_VEL
LIN {X 0,Y 199.861,Z 188.568,A -85,B 0,C 180,E1 -21612.18,E2 -21612.18} C_VEL
LIN {X 0,Y 199.786,Z 188.586,A -85,B 0,C 180,E1 -21616.345,E2 -21616.345} C_VEL
LIN {X 0,Y 199.674,Z 188.613,A -85,B 0,C 180,E1 -21620.608,E2 -21620.608} C_VEL
LIN {X 0,Y 199.664,Z 188.599,A -85,B 0,C 180,E1 -21624.986,E2 -21624.986} C_VEL
LIN {X 0,Y 199.664,Z 188.598,A -85,B 0,C 180,E1 -21629.524,E2 -21629.524} C_VEL
LIN {X 0,Y 199.671,Z 188.613,A -85,B 0,C 180,E1 -21632.355,E2 -21632.355} C_VEL
LIN {X 0,Y 199.622,Z 188.563,A -85,B 0,C 180,E1 -21636.763,E2 -21636.763} C_VEL
LIN {X 0,Y 199.606,Z 188.593,A -85,B 0,C 180,E1 -21639.329,E2 -21639.329} C_VEL
LIN {X 0,Y 199.594,Z 188.663,A -85,B 0,C 180,E1 -21644.684,E2 -21644.684} C_VEL
LIN {X 0,Y 200.498,Z 191.751,A -85,B 0,C 180,E1 -21646.739,E2 -21646.739} C_VEL
LIN {X 0,Y 202.858,Z 195.959,A -85,B 0,C 180,E1 -21647.665,E2 -21647.665} C_VEL
LIN {X 0,Y 209.069,Z 206.67,A -85,B 0,C 180,E1 -21649.669,E2 -21649.669} C_VEL
LIN {X 0,Y 214.813,Z 217.83,A -85,B 0,C 180,E1 -21651.424,E2 -21651.424} C_VEL
LIN {X 0,Y 215.703,Z 221.487,A -85,B 0,C 180,E1 -21651.764,E2 -21651.764} C_VEL
LIN {X 0,Y 216.243,Z 234.684,A -85,B 0,C 180,E1 -21652.42,E2 -21652.42} C_VEL
LIN {X 0,Y 217.009,Z 238.438,A -85,B 0,C 180,E1 -21652.729,E2 -21652.729} C_VEL
LIN {X 0,Y 218.708,Z 243.244,A -85,B 0,C 180,E1 -21653.259,E2 -21653.259} C_VEL
LIN {X 0,Y 219.073,Z 246.525,A -85,B 0,C 180,E1 -21653.461,E2 -21653.461} C_VEL
LIN {X 0,Y 216.463,Z 300.152,A -85,B 0,C 180,E1 -21655.166,E2 -21655.166} C_VEL
LIN {X 0,Y 214.991,Z 313.255,A -85,B 0,C 180,E1 -21655.89,E2 -21655.89} C_VEL
LIN {X 0,Y 213.001,Z 325.277,A -85,B 0,C 180,E1 -21656.874,E2 -21656.874} C_VEL
LIN {X 0,Y 210.539,Z 337.453,A -85,B 0,C 180,E1 -21658.281,E2 -21658.281} C_VEL
LIN {X 0,Y 207.674,Z 348.996,A -85,B 0,C 180,E1 -21660.055,E2 -21660.055} C_VEL
LIN {X 0,Y 204.627,Z 359.39,A -85,B 0,C 180,E1 -21662.098,E2 -21662.098} C_VEL
LIN {X 0,Y 201.889,Z 367.885,A -85,B 0,C 180,E1 -21664.206,E2 -21664.206} C_VEL
LIN {X 0,Y 199.489,Z 375.458,A -85,B 0,C 180,E1 -21666.55,E2 -21666.55} C_VEL
LIN {X 0,Y 196.617,Z 383.376,A -85,B 0,C 180,E1 -21669.603,E2 -21669.603} C_VEL
LIN {X 0,Y 193.926,Z 390.433,A -85,B 0,C 180,E1 -21673.146,E2 -21673.146} C_VEL
LIN {X 0,Y 192.306,Z 395.127,A -85,B 0,C 180,E1 -21676.257,E2 -21676.257} C_VEL
LIN {X 0,Y 191.157,Z 398.711,A -85,B 0,C 180,E1 -21679.407,E2 -21679.407} C_VEL
LIN {X 0,Y 190.656,Z 400.558,A -85,B 0,C 180,E1 -21681.52,E2 -21681.52} C_VEL
LIN {X 0,Y 190.355,Z 401.943,A -85,B 0,C 180,E1 -21683.64,E2 -21683.64} C_VEL
LIN {X 0,Y 190.144,Z 403.152,A -85,B 0,C 180,E1 -21686.343,E2 -21686.343} C_VEL
LIN {X 0,Y 190.154,Z 403.743,A -85,B 0,C 180,E1 -21689.999,E2 -21689.999} C_VEL
LIN {X 0,Y 190.143,Z 403.131,A -85,B 0,C 180,E1 -21693.655,E2 -21693.655} C_VEL
LIN {X 0,Y 190.355,Z 401.914,A -85,B 0,C 180,E1 -21696.358,E2 -21696.358} C_VEL
LIN {X 0,Y 190.657,Z 400.516,A -85,B 0,C 180,E1 -21698.478,E2 -21698.478} C_VEL
LIN {X 0,Y 191.491,Z 397.584,A -85,B 0,C 180,E1 -21701.644,E2 -21701.644} C_VEL
LIN {X 0,Y 192.77,Z 393.616,A -85,B 0,C 180,E1 -21704.784,E2 -21704.784} C_VEL
LIN {X 0,Y 194.995,Z 387.515,A -85,B 0,C 180,E1 -21708.382,E2 -21708.382} C_VEL
LIN {X 0,Y 197.435,Z 380.85,A -85,B 0,C 180,E1 -21711.398,E2 -21711.398} C_VEL
LIN {X 0,Y 200.119,Z 373.186,A -85,B 0,C 180,E1 -21714.145,E2 -21714.145} C_VEL
LIN {X 0,Y 203.029,Z 364.095,A -85,B 0,C 180,E1 -21716.742,E2 -21716.742} C_VEL
LIN {X 0,Y 206.253,Z 353.609,A -85,B 0,C 180,E1 -21719.048,E2 -21719.048} C_VEL
LIN {X 0,Y 209.004,Z 343.229,A -85,B 0,C 180,E1 -21720.849,E2 -21720.849} C_VEL
LIN {X 0,Y 211.671,Z 331.838,A -85,B 0,C 180,E1 -21722.369,E2 -21722.369} C_VEL
LIN {X 0,Y 213.779,Z 320.098,A -85,B 0,C 180,E1 -21723.551,E2 -21723.551} C_VEL
LIN {X 0,Y 215.692,Z 306.573,A -85,B 0,C 180,E1 -21724.478,E2 -21724.478} C_VEL
LIN {X 0,Y 216.703,Z 293.995,A -85,B 0,C 180,E1 -21725.027,E2 -21725.027} C_VEL
LIN {X 0,Y 218.946,Z 245.695,A -85,B 0,C 180,E1 -21726.526,E2 -21726.526} C_VEL
LIN {X 0,Y 218.083,Z 241.471,A -85,B 0,C 180,E1 -21726.864,E2 -21726.864} C_VEL
LIN {X 0,Y 211.994,Z 226.524,A -85,B 0,C 180,E1 -21728.736,E2 -21728.736} C_VEL
LIN {X 0,Y 205.875,Z 213.694,A -85,B 0,C 180,E1 -21730.687,E2 -21730.687} C_VEL
LIN {X 0,Y 200.306,Z 203.721,A -85,B 0,C 180,E1 -21732.539,E2 -21732.539} C_VEL
LIN {X 0,Y 195.437,Z 195.65,A -85,B 0,C 180,E1 -21734.263,E2 -21734.263} C_VEL
LIN {X 0,Y 193.135,Z 191.656,A -85,B 0,C 180,E1 -21735.259,E2 -21735.259} C_VEL
LIN {X 0,Y 192.503,Z 189.55,A -85,B 0,C 180,E1 -21736.737,E2 -21736.737} C_VEL
LIN {X 0,Y 192.545,Z 189.453,A -85,B 0,C 180,E1 -21741.647,E2 -21741.647} C_VEL
LIN {X 0,Y 192.591,Z 189.481,A -85,B 0,C 180,E1 -21746.813,E2 -21746.813} C_VEL
LIN {X 0,Y 192.655,Z 189.475,A -85,B 0,C 180,E1 -21751.69,E2 -21751.69} C_VEL
LIN {X 0,Y 192.678,Z 189.464,A -85,B 0,C 180,E1 -21756.345,E2 -21756.345} C_VEL
LIN {X 0,Y 192.723,Z 189.457,A -85,B 0,C 180,E1 -21761.459,E2 -21761.459} C_VEL
LIN {X 0,Y 192.745,Z 189.477,A -85,B 0,C 180,E1 -21765.212,E2 -21765.212} C_VEL
LIN {X 0,Y 192.975,Z 189.426,A -85,B 0,C 180,E1 -21769.508,E2 -21769.508} C_VEL
LIN {X 0,Y 193.054,Z 189.437,A -85,B 0,C 180,E1 -21771.627,E2 -21771.627} C_VEL
LIN {X 0,Y 193.253,Z 189.409,A -85,B 0,C 180,E1 -21777.916,E2 -21777.916} C_VEL
LIN {X 0,Y 193.435,Z 189.383,A -85,B 0,C 180,E1 -21780,E2 -21780} C_VEL
LIN {X 0,Y 192.965,Z 189.433,A -85,B 0,C 180,E1 -21784.177,E2 -21784.177} C_VEL
LIN {X 0,Y 193.054,Z 189.412,A -85,B 0,C 180,E1 -21788.373,E2 -21788.373} C_VEL
LIN {X 0,Y 192.845,Z 189.462,A -85,B 0,C 180,E1 -21792.631,E2 -21792.631} C_VEL
LIN {X 0,Y 192.775,Z 189.471,A -85,B 0,C 180,E1 -21798.587,E2 -21798.587} C_VEL
LIN {X 0,Y 192.659,Z 189.483,A -85,B 0,C 180,E1 -21804.225,E2 -21804.225} C_VEL
LIN {X 0,Y 192.645,Z 189.475,A -85,B 0,C 180,E1 -21808.893,E2 -21808.893} C_VEL
LIN {X 0,Y 192.594,Z 189.448,A -85,B 0,C 180,E1 -21813.187,E2 -21813.187} C_VEL
LIN {X 0,Y 192.547,Z 189.475,A -85,B 0,C 180,E1 -21818.353,E2 -21818.353} C_VEL
LIN {X 0,Y 192.485,Z 189.464,A -85,B 0,C 180,E1 -21823.096,E2 -21823.096} C_VEL
LIN {X 0,Y 192.585,Z 189.834,A -85,B 0,C 180,E1 -21824.522,E2 -21824.522} C_VEL
LIN {X 0,Y 192.922,Z 191.048,A -85,B 0,C 180,E1 -21824.926,E2 -21824.926} C_VEL
LIN {X 0,Y 194.556,Z 193.628,A -85,B 0,C 180,E1 -21825.556,E2 -21825.556} C_VEL
LIN {X 0,Y 195.728,Z 194.995,A -85,B 0,C 180,E1 -21825.961,E2 -21825.961} C_VEL
LIN {X 0,Y 198.031,Z 198.458,A -85,B 0,C 180,E1 -21826.773,E2 -21826.773} C_VEL
LIN {X 0,Y 203.884,Z 208.176,A -85,B 0,C 180,E1 -21828.753,E2 -21828.753} C_VEL
LIN {X 0,Y 210.504,Z 221.081,A -85,B 0,C 180,E1 -21830.878,E2 -21830.878} C_VEL
LIN {X 0,Y 217.325,Z 236.589,A -85,B 0,C 180,E1 -21832.962,E2 -21832.962} C_VEL
LIN {X 0,Y 219.147,Z 241.518,A -85,B 0,C 180,E1 -21833.519,E2 -21833.519} C_VEL
